	VAR robtarget Openhole_5522 := [[482.14, -9.61, 178.45], [0.078704, 0.702713, 0.693768, -0.136696], [0,0,0,0], [9E9, 9E9, 9E9, 9E9, 9E9, 9E9]];
	VAR robtarget Openhole_5523 := [[481.64, -9.62, 178.5], [0.077135, 0.702887, 0.694058, -0.135217], [0,0,0,0], [9E9, 9E9, 9E9, 9E9, 9E9, 9E9]];
	VAR robtarget Openhole_5524 := [[476.67, -9.77, 178.99], [0.061718, 0.704408, 0.696901, -0.119702], [0,0,0,0], [9E9, 9E9, 9E9, 9E9, 9E9, 9E9]];
	VAR robtarget Openhole_5525 := [[472.72, -10.2, 179.44], [0.050233, 0.70532, 0.699112, -0.106028], [0,0,0,0], [9E9, 9E9, 9E9, 9E9, 9E9, 9E9]];
	VAR robtarget Openhole_5526 := [[469.79, -10.75, 179.79], [0.042383, 0.705835, 0.700704, -0.094942], [0,0,0,0], [9E9, 9E9, 9E9, 9E9, 9E9, 9E9]];
	VAR robtarget Openhole_5527 := [[466.45, -11.71, 180.22], [0.034434, 0.706268, 0.702451, -0.081013], [0,0,0,0], [9E9, 9E9, 9E9, 9E9, 9E9, 9E9]];
	VAR robtarget Openhole_5528 := [[465.52, -12.04, 180.33], [0.0324, 0.706364, 0.702917, -0.076862], [0,0,0,0], [9E9, 9E9, 9E9, 9E9, 9E9, 9E9]];
	VAR robtarget Openhole_5529 := [[465.05, -12.22, 180.39], [0.031455, 0.706407, 0.703145, -0.074747], [0,0,0,0], [9E9, 9E9, 9E9, 9E9, 9E9, 9E9]];
	VAR robtarget Openhole_5530 := [[463.68, -12.81, 180.56], [0.028831, 0.706519, 0.703802, -0.068286], [0,0,0,0], [9E9, 9E9, 9E9, 9E9, 9E9, 9E9]];
	VAR robtarget Openhole_5531 := [[463.23, -13.02, 180.62], [0.028028, 0.706551, 0.704011, -0.066095], [0,0,0,0], [9E9, 9E9, 9E9, 9E9, 9E9, 9E9]];
	VAR robtarget Openhole_5532 := [[461.04, -14.18, 180.88], [0.024524, 0.706681, 0.704972, -0.05491], [0,0,0,0], [9E9, 9E9, 9E9, 9E9, 9E9, 9E9]];
	VAR robtarget Openhole_5533 := [[460.18, -14.69, 180.97], [0.023348, 0.706721, 0.705312, -0.050345], [0,0,0,0], [9E9, 9E9, 9E9, 9E9, 9E9, 9E9]];
	VAR robtarget Openhole_5534 := [[459.34, -15.23, 181.06], [0.022345, 0.706754, 0.705627, -0.045724], [0,0,0,0], [9E9, 9E9, 9E9, 9E9, 9E9, 9E9]];
	VAR robtarget Openhole_5535 := [[458.92, -15.49, 181.1], [0.021792, 0.706771, 0.705772, -0.04342], [0,0,0,0], [9E9, 9E9, 9E9, 9E9, 9E9, 9E9]];
	VAR robtarget Openhole_5536 := [[458.49, -15.74, 181.13], [0.021166, 0.70679, 0.70591, -0.041131], [0,0,0,0], [9E9, 9E9, 9E9, 9E9, 9E9, 9E9]];
	VAR robtarget Openhole_5537 := [[457.6, -16.2, 181.2], [0.019722, 0.706832, 0.706159, -0.036599], [0,0,0,0], [9E9, 9E9, 9E9, 9E9, 9E9, 9E9]];
	VAR robtarget Openhole_5538 := [[457.02, -16.45, 181.23], [0.018633, 0.706861, 0.706298, -0.033803], [0,0,0,0], [9E9, 9E9, 9E9, 9E9, 9E9, 9E9]];
	VAR robtarget Openhole_5539 := [[454.58, -16.45, 181.29], [0.010319, 0.707031, 0.706646, -0.025537], [0,0,0,0], [9E9, 9E9, 9E9, 9E9, 9E9, 9E9]];
	VAR robtarget Openhole_5540 := [[454.01, -15.03, 181.24], [0.003545, 0.707098, 0.706535, -0.028428], [0,0,0,0], [9E9, 9E9, 9E9, 9E9, 9E9, 9E9]];
	VAR robtarget Openhole_5541 := [[456.45, -15.03, 181.15], [0.011872, 0.707007, 0.706154, -0.036692], [0,0,0,0], [9E9, 9E9, 9E9, 9E9, 9E9, 9E9]];
	VAR robtarget Openhole_5542 := [[457.91, -14.13, 181.02], [0.013741, 0.706973, 0.705696, -0.044638], [0,0,0,0], [9E9, 9E9, 9E9, 9E9, 9E9, 9E9]];
	VAR robtarget Openhole_5543 := [[458.76, -13.61, 180.93], [0.014897, 0.70695, 0.705391, -0.049232], [0,0,0,0], [9E9, 9E9, 9E9, 9E9, 9E9, 9E9]];
	VAR robtarget Openhole_5544 := [[459.2, -13.37, 180.89], [0.015574, 0.706935, 0.705229, -0.051497], [0,0,0,0], [9E9, 9E9, 9E9, 9E9, 9E9, 9E9]];
	VAR robtarget Openhole_5545 := [[459.64, -13.14, 180.84], [0.016297, 0.706919, 0.705061, -0.053745], [0,0,0,0], [9E9, 9E9, 9E9, 9E9, 9E9, 9E9]];
	VAR robtarget Openhole_5546 := [[460.54, -12.71, 180.74], [0.017862, 0.706881, 0.704708, -0.05819], [0,0,0,0], [9E9, 9E9, 9E9, 9E9, 9E9, 9E9]];
	VAR robtarget Openhole_5547 := [[461.9, -12.1, 180.58], [0.020434, 0.706811, 0.704136, -0.064748], [0,0,0,0], [9E9, 9E9, 9E9, 9E9, 9E9, 9E9]];
	VAR robtarget Openhole_5548 := [[463.74, -11.36, 180.36], [0.024178, 0.706693, 0.703297, -0.073302], [0,0,0,0], [9E9, 9E9, 9E9, 9E9, 9E9, 9E9]];
	VAR robtarget Openhole_5549 := [[466.57, -10.43, 180], [0.030537, 0.706447, 0.701901, -0.085647], [0,0,0,0], [9E9, 9E9, 9E9, 9E9, 9E9, 9E9]];
	VAR robtarget Openhole_5550 := [[468.97, -9.8, 179.68], [0.036475, 0.706165, 0.700635, -0.095449], [0,0,0,0], [9E9, 9E9, 9E9, 9E9, 9E9, 9E9]];
	VAR robtarget Openhole_5551 := [[472.87, -9.09, 179.17], [0.047062, 0.705539, 0.698476, -0.110139], [0,0,0,0], [9E9, 9E9, 9E9, 9E9, 9E9, 9E9]];
	VAR robtarget Openhole_5552 := [[477.32, -8.67, 178.63], [0.060222, 0.704538, 0.695928, -0.125238], [0,0,0,0], [9E9, 9E9, 9E9, 9E9, 9E9, 9E9]];
	VAR robtarget Openhole_5553 := [[481.79, -8.56, 178.15], [0.074227, 0.7032, 0.693312, -0.13899], [0,0,0,0], [9E9, 9E9, 9E9, 9E9, 9E9, 9E9]];
	VAR robtarget Openhole_5554 := [[482.29, -8.56, 178.1], [0.075808, 0.703031, 0.693017, -0.140454], [0,0,0,0], [9E9, 9E9, 9E9, 9E9, 9E9, 9E9]];
	VAR robtarget Openhole_5555 := [[490.75, -8.89, 177.38], [0.102945, 0.699573, 0.687924, -0.163586], [0,0,0,0], [9E9, 9E9, 9E9, 9E9, 9E9, 9E9]];
	VAR robtarget Openhole_5556 := [[499.22, -9.25, 176.73], [0.128731, 0.69529, 0.682463, -0.185054], [0,0,0,0], [9E9, 9E9, 9E9, 9E9, 9E9, 9E9]];
	VAR robtarget Openhole_5557 := [[500.21, -9.26, 176.64], [0.131553, 0.694762, 0.681773, -0.187578], [0,0,0,0], [9E9, 9E9, 9E9, 9E9, 9E9, 9E9]];
	VAR robtarget Openhole_5558 := [[500.71, -9.26, 176.59], [0.132933, 0.694499, 0.681421, -0.188853], [0,0,0,0], [9E9, 9E9, 9E9, 9E9, 9E9, 9E9]];
	VAR robtarget Openhole_5559 := [[503.19, -9.2, 176.33], [0.139644, 0.693181, 0.679622, -0.195227], [0,0,0,0], [9E9, 9E9, 9E9, 9E9, 9E9, 9E9]];
	VAR robtarget Openhole_5560 := [[503.69, -9.17, 176.27], [0.1409, 0.692927, 0.679243, -0.196542], [0,0,0,0], [9E9, 9E9, 9E9, 9E9, 9E9, 9E9]];
	VAR robtarget Openhole_5561 := [[504.33, -9.15, 176.19], [0.142564, 0.692586, 0.678764, -0.198192], [0,0,0,0], [9E9, 9E9, 9E9, 9E9, 9E9, 9E9]];
	VAR robtarget Openhole_5562 := [[509.33, -9.15, 175.72], [0.183051, 0.683002, 0.683002, -0.183051], [0,0,0,0], [9E9, 9E9, 9E9, 9E9, 9E9, 9E9]];
	VAR robtarget Openhole_5563 := [[536.33, -9.15, 175.63], [0.183051, 0.683002, 0.683002, -0.183051], [0,0,0,0], [9E9, 9E9, 9E9, 9E9, 9E9, 9E9]];
	VAR robtarget Openhole_5564 := [[536.33, -8.27, 175.13], [0.183051, 0.683002, 0.683002, -0.183051], [0,0,0,0], [9E9, 9E9, 9E9, 9E9, 9E9, 9E9]];
	VAR robtarget Openhole_5565 := [[524.33, -8.27, 175.17], [0.183051, 0.683002, 0.683002, -0.183051], [0,0,0,0], [9E9, 9E9, 9E9, 9E9, 9E9, 9E9]];
	VAR robtarget Openhole_5566 := [[509.33, -8.28, 175.21], [0.183051, 0.683002, 0.683002, -0.183051], [0,0,0,0], [9E9, 9E9, 9E9, 9E9, 9E9, 9E9]];
	VAR robtarget Openhole_5567 := [[504.35, -8.28, 175.73], [0.140085, 0.693092, 0.678014, -0.20074], [0,0,0,0], [9E9, 9E9, 9E9, 9E9, 9E9, 9E9]];
	VAR robtarget Openhole_5568 := [[503.83, -8.3, 175.8], [0.138746, 0.693361, 0.678412, -0.199393], [0,0,0,0], [9E9, 9E9, 9E9, 9E9, 9E9, 9E9]];
	VAR robtarget Openhole_5569 := [[501.35, -8.33, 176.06], [0.131956, 0.694685, 0.68021, -0.193171], [0,0,0,0], [9E9, 9E9, 9E9, 9E9, 9E9, 9E9]];
	VAR robtarget Openhole_5570 := [[500.85, -8.32, 176.11], [0.13055, 0.694951, 0.680559, -0.191937], [0,0,0,0], [9E9, 9E9, 9E9, 9E9, 9E9, 9E9]];
	VAR robtarget Openhole_5571 := [[493.88, -7.98, 176.68], [0.10947, 0.698582, 0.685143, -0.174867], [0,0,0,0], [9E9, 9E9, 9E9, 9E9, 9E9, 9E9]];
	VAR robtarget Openhole_5572 := [[483.94, -7.4, 177.55], [0.077321, 0.702867, 0.691248, -0.148916], [0,0,0,0], [9E9, 9E9, 9E9, 9E9, 9E9, 9E9]];
	VAR robtarget Openhole_5573 := [[480.96, -7.35, 177.87], [0.0677, 0.703858, 0.69304, -0.140343], [0,0,0,0], [9E9, 9E9, 9E9, 9E9, 9E9, 9E9]];
	VAR robtarget Openhole_5574 := [[480.46, -7.35, 177.92], [0.066114, 0.704009, 0.693337, -0.138866], [0,0,0,0], [9E9, 9E9, 9E9, 9E9, 9E9, 9E9]];
	VAR robtarget Openhole_5575 := [[476, -7.51, 178.47], [0.052157, 0.705181, 0.695985, -0.12492], [0,0,0,0], [9E9, 9E9, 9E9, 9E9, 9E9, 9E9]];
	VAR robtarget Openhole_5576 := [[471.56, -7.98, 179.06], [0.039093, 0.706025, 0.698557, -0.109628], [0,0,0,0], [9E9, 9E9, 9E9, 9E9, 9E9, 9E9]];
	VAR robtarget Openhole_5577 := [[467.18, -8.8, 179.67], [0.027176, 0.706584, 0.700967, -0.092983], [0,0,0,0], [9E9, 9E9, 9E9, 9E9, 9E9, 9E9]];
	VAR robtarget Openhole_5578 := [[464.77, -9.39, 179.99], [0.021046, 0.706794, 0.702192, -0.083224], [0,0,0,0], [9E9, 9E9, 9E9, 9E9, 9E9, 9E9]];
	VAR robtarget Openhole_5579 := [[459.06, -11.07, 180.68], [0.007315, 0.707069, 0.704662, -0.058745], [0,0,0,0], [9E9, 9E9, 9E9, 9E9, 9E9, 9E9]];
	VAR robtarget Openhole_5580 := [[458.11, -11.38, 180.78], [0.005116, 0.707088, 0.704999, -0.05456], [0,0,0,0], [9E9, 9E9, 9E9, 9E9, 9E9, 9E9]];
	VAR robtarget Openhole_5581 := [[457.17, -11.7, 180.87], [0.00302, 0.7071, 0.705315, -0.05031], [0,0,0,0], [9E9, 9E9, 9E9, 9E9, 9E9, 9E9]];
	VAR robtarget Openhole_5582 := [[456.7, -11.89, 180.92], [0.002058, 0.707104, 0.705466, -0.048142], [0,0,0,0], [9E9, 9E9, 9E9, 9E9, 9E9, 9E9]];
	VAR robtarget Openhole_5583 := [[456.25, -12.09, 180.96], [0.001205, 0.707106, 0.705614, -0.045926], [0,0,0,0], [9E9, 9E9, 9E9, 9E9, 9E9, 9E9]];
	VAR robtarget Openhole_5584 := [[455.8, -12.3, 181], [0.000391, 0.707107, 0.705756, -0.043694], [0,0,0,0], [9E9, 9E9, 9E9, 9E9, 9E9, 9E9]];
	VAR robtarget Openhole_5585 := [[455.36, -12.53, 181.05], [-0.000349, 0.707107, 0.705892, -0.041433], [0,0,0,0], [9E9, 9E9, 9E9, 9E9, 9E9, 9E9]];
	VAR robtarget Openhole_5586 := [[454.83, -12.87, 181.1], [-0.001006, 0.707106, 0.706058, -0.038495], [0,0,0,0], [9E9, 9E9, 9E9, 9E9, 9E9, 9E9]];
	VAR robtarget Openhole_5587 := [[445.25, -11.83, 181.71], [-0.03715, 0.70613, 0.707042, -0.009558], [0,0,0,0], [9E9, 9E9, 9E9, 9E9, 9E9, 9E9]];
	VAR robtarget Openhole_5588 := [[444.72, -11.69, 181.75], [-0.039438, 0.706006, 0.707059, -0.008218], [0,0,0,0], [9E9, 9E9, 9E9, 9E9, 9E9, 9E9]];
	VAR robtarget Openhole_5589 := [[444.22, -11.62, 181.79], [-0.041326, 0.705898, 0.707075, -0.006749], [0,0,0,0], [9E9, 9E9, 9E9, 9E9, 9E9, 9E9]];
	VAR robtarget Openhole_5590 := [[443.23, -11.52, 181.86], [-0.045015, 0.705673, 0.707097, -0.003709], [0,0,0,0], [9E9, 9E9, 9E9, 9E9, 9E9, 9E9]];
	VAR robtarget Openhole_5591 := [[442.24, -11.45, 181.94], [-0.048615, 0.705434, 0.707107, -0.000574], [0,0,0,0], [9E9, 9E9, 9E9, 9E9, 9E9, 9E9]];
	VAR robtarget Openhole_5592 := [[441.74, -11.43, 181.98], [-0.050381, 0.70531, 0.707106, 0.001028], [0,0,0,0], [9E9, 9E9, 9E9, 9E9, 9E9, 9E9]];
	VAR robtarget Openhole_5593 := [[431.77, -11.25, 182.74], [-0.08402, 0.702097, 0.706286, 0.03406], [0,0,0,0], [9E9, 9E9, 9E9, 9E9, 9E9, 9E9]];
	VAR robtarget Openhole_5594 := [[431.27, -11.25, 182.77], [-0.085634, 0.701902, 0.706204, 0.035729], [0,0,0,0], [9E9, 9E9, 9E9, 9E9, 9E9, 9E9]];
	VAR robtarget Openhole_5595 := [[407.33, -11.81, 184.34], [-0.156518, 0.689567, 0.697978, 0.113254], [0,0,0,0], [9E9, 9E9, 9E9, 9E9, 9E9, 9E9]];
	VAR robtarget Openhole_5596 := [[396.35, -12.23, 184.89], [-0.184529, 0.682605, 0.69195, 0.145619], [0,0,0,0], [9E9, 9E9, 9E9, 9E9, 9E9, 9E9]];
	VAR robtarget Openhole_5597 := [[394.34, -12.34, 184.96], [-0.189276, 0.681304, 0.690716, 0.151363], [0,0,0,0], [9E9, 9E9, 9E9, 9E9, 9E9, 9E9]];
	VAR robtarget Openhole_5598 := [[389.36, -12.34, 185.28], [-0.201409, 0.677816, 0.687741, 0.164354], [0,0,0,0], [9E9, 9E9, 9E9, 9E9, 9E9, 9E9]];
	VAR robtarget Openhole_5599 := [[362.36, -12.34, 185.37], [-0.183051, 0.683002, 0.683002, 0.183051], [0,0,0,0], [9E9, 9E9, 9E9, 9E9, 9E9, 9E9]];
	VAR robtarget Openhole_5600 := [[362.36, -13.23, 184.86], [-0.183051, 0.683002, 0.683002, 0.183051], [0,0,0,0], [9E9, 9E9, 9E9, 9E9, 9E9, 9E9]];
	VAR robtarget Openhole_5601 := [[374.36, -13.23, 184.82], [-0.183051, 0.683002, 0.683002, 0.183051], [0,0,0,0], [9E9, 9E9, 9E9, 9E9, 9E9, 9E9]];
	VAR robtarget Openhole_5602 := [[389.36, -13.23, 184.77], [-0.198916, 0.678552, 0.687133, 0.166878], [0,0,0,0], [9E9, 9E9, 9E9, 9E9, 9E9, 9E9]];
	VAR robtarget Openhole_5603 := [[394.33, -13.23, 184.49], [-0.186724, 0.682007, 0.690143, 0.153955], [0,0,0,0], [9E9, 9E9, 9E9, 9E9, 9E9, 9E9]];
	VAR robtarget Openhole_5604 := [[404.34, -12.8, 184.12], [-0.161764, 0.688355, 0.695969, 0.125011], [0,0,0,0], [9E9, 9E9, 9E9, 9E9, 9E9, 9E9]];
	VAR robtarget Openhole_5605 := [[421.81, -12.49, 183.16], [-0.111659, 0.698235, 0.703558, 0.070753], [0,0,0,0], [9E9, 9E9, 9E9, 9E9, 9E9, 9E9]];
	VAR robtarget Openhole_5606 := [[427.8, -12.45, 182.78], [-0.092876, 0.700981, 0.70525, 0.051205], [0,0,0,0], [9E9, 9E9, 9E9, 9E9, 9E9, 9E9]];
	VAR robtarget Openhole_5607 := [[428.3, -12.46, 182.75], [-0.09127, 0.701192, 0.705367, 0.049569], [0,0,0,0], [9E9, 9E9, 9E9, 9E9, 9E9, 9E9]];
	VAR robtarget Openhole_5608 := [[434.78, -12.62, 182.32], [-0.069589, 0.703674, 0.70653, 0.028563], [0,0,0,0], [9E9, 9E9, 9E9, 9E9, 9E9, 9E9]];
	VAR robtarget Openhole_5609 := [[440.25, -13.05, 181.95], [-0.049924, 0.705342, 0.707013, 0.011547], [0,0,0,0], [9E9, 9E9, 9E9, 9E9, 9E9, 9E9]];
	VAR robtarget Openhole_5610 := [[442.74, -13.1, 181.8], [-0.041319, 0.705899, 0.707099, 0.003283], [0,0,0,0], [9E9, 9E9, 9E9, 9E9, 9E9, 9E9]];
	VAR robtarget Openhole_5611 := [[443.44, -13.31, 181.75], [-0.038283, 0.70607, 0.707105, 0.001638], [0,0,0,0], [9E9, 9E9, 9E9, 9E9, 9E9, 9E9]];
	VAR robtarget Openhole_5612 := [[445.21, -13.31, 181.65], [-0.03227, 0.70637, 0.707093, -0.004388], [0,0,0,0], [9E9, 9E9, 9E9, 9E9, 9E9, 9E9]];
	VAR robtarget Openhole_5613 := [[444.28, -14.54, 181.64], [-0.031215, 0.706417, 0.707101, 0.002931], [0,0,0,0], [9E9, 9E9, 9E9, 9E9, 9E9, 9E9]];
	VAR robtarget Openhole_5614 := [[442.51, -14.54, 181.72], [-0.037224, 0.706126, 0.70705, 0.008951], [0,0,0,0], [9E9, 9E9, 9E9, 9E9, 9E9, 9E9]];
	VAR robtarget Openhole_5615 := [[441.98, -14.53, 181.74], [-0.039072, 0.706026, 0.707026, 0.010719], [0,0,0,0], [9E9, 9E9, 9E9, 9E9, 9E9, 9E9]];
	VAR robtarget Openhole_5616 := [[440.98, -14.49, 181.79], [-0.042583, 0.705823, 0.706969, 0.013957], [0,0,0,0], [9E9, 9E9, 9E9, 9E9, 9E9, 9E9]];
	VAR robtarget Openhole_5617 := [[439.98, -14.49, 181.83], [-0.045964, 0.705611, 0.706895, 0.017319], [0,0,0,0], [9E9, 9E9, 9E9, 9E9, 9E9, 9E9]];
	VAR robtarget Openhole_5618 := [[439.48, -14.47, 181.85], [-0.04768, 0.705497, 0.706852, 0.01897], [0,0,0,0], [9E9, 9E9, 9E9, 9E9, 9E9, 9E9]];
	VAR robtarget Openhole_5619 := [[438.98, -14.45, 181.88], [-0.049444, 0.705376, 0.706808, 0.020564], [0,0,0,0], [9E9, 9E9, 9E9, 9E9, 9E9, 9E9]];
	VAR robtarget Openhole_5620 := [[438.48, -14.4, 181.9], [-0.051258, 0.705247, 0.706761, 0.022097], [0,0,0,0], [9E9, 9E9, 9E9, 9E9, 9E9, 9E9]];
	VAR robtarget Openhole_5621 := [[433.03, -13.83, 182.24], [-0.071327, 0.7035, 0.70606, 0.038469], [0,0,0,0], [9E9, 9E9, 9E9, 9E9, 9E9, 9E9]];
	VAR robtarget Openhole_5622 := [[426.54, -13.59, 182.61], [-0.093145, 0.700945, 0.704635, 0.05907], [0,0,0,0], [9E9, 9E9, 9E9, 9E9, 9E9, 9E9]];
	VAR robtarget Openhole_5623 := [[419.55, -13.55, 182.99], [-0.115196, 0.69766, 0.702409, 0.08137], [0,0,0,0], [9E9, 9E9, 9E9, 9E9, 9E9, 9E9]];
	VAR robtarget Openhole_5624 := [[419.05, -13.55, 183.02], [-0.116726, 0.697406, 0.702225, 0.082945], [0,0,0,0], [9E9, 9E9, 9E9, 9E9, 9E9, 9E9]];
	VAR robtarget Openhole_5625 := [[404.07, -13.73, 183.73], [-0.159674, 0.688843, 0.695311, 0.128617], [0,0,0,0], [9E9, 9E9, 9E9, 9E9, 9E9, 9E9]];
	VAR robtarget Openhole_5626 := [[394.35, -14.11, 184.02], [-0.18411, 0.682718, 0.689575, 0.156483], [0,0,0,0], [9E9, 9E9, 9E9, 9E9, 9E9, 9E9]];
	VAR robtarget Openhole_5627 := [[389.36, -14.11, 184.26], [-0.19642, 0.679279, 0.686516, 0.1694], [0,0,0,0], [9E9, 9E9, 9E9, 9E9, 9E9, 9E9]];
	VAR robtarget Openhole_5628 := [[362.36, -14.11, 184.35], [-0.183051, 0.683002, 0.683002, 0.183051], [0,0,0,0], [9E9, 9E9, 9E9, 9E9, 9E9, 9E9]];
	VAR robtarget Openhole_5629 := [[362.35, -15.07, 183.79], [-0.183051, 0.683002, 0.683002, 0.183051], [0,0,0,0], [9E9, 9E9, 9E9, 9E9, 9E9, 9E9]];
	VAR robtarget Openhole_5630 := [[389.35, -15.07, 183.7], [-0.193687, 0.680063, 0.68583, 0.172155], [0,0,0,0], [9E9, 9E9, 9E9, 9E9, 9E9, 9E9]];
	VAR robtarget Openhole_5631 := [[394.35, -15.07, 183.51], [-0.181307, 0.683467, 0.688928, 0.159306], [0,0,0,0], [9E9, 9E9, 9E9, 9E9, 9E9, 9E9]];
	VAR robtarget Openhole_5632 := [[404.04, -14.7, 183.31], [-0.15678, 0.689507, 0.694738, 0.131678], [0,0,0,0], [9E9, 9E9, 9E9, 9E9, 9E9, 9E9]];
	VAR robtarget Openhole_5633 := [[413.54, -14.6, 182.95], [-0.12998, 0.695058, 0.699507, 0.10339], [0,0,0,0], [9E9, 9E9, 9E9, 9E9, 9E9, 9E9]];
	VAR robtarget Openhole_5634 := [[414.04, -14.6, 182.93], [-0.128498, 0.695333, 0.69973, 0.101869], [0,0,0,0], [9E9, 9E9, 9E9, 9E9, 9E9, 9E9]];
	VAR robtarget Openhole_5635 := [[427.52, -14.77, 182.32], [-0.086129, 0.701842, 0.704577, 0.059757], [0,0,0,0], [9E9, 9E9, 9E9, 9E9, 9E9, 9E9]];
	VAR robtarget Openhole_5636 := [[434, -15.12, 182], [-0.063775, 0.704225, 0.706, 0.039544], [0,0,0,0], [9E9, 9E9, 9E9, 9E9, 9E9, 9E9]];
	VAR robtarget Openhole_5637 := [[437.48, -15.49, 181.83], [-0.050954, 0.705269, 0.706505, 0.029156], [0,0,0,0], [9E9, 9E9, 9E9, 9E9, 9E9, 9E9]];
	VAR robtarget Openhole_5638 := [[438.47, -15.58, 181.78], [-0.047326, 0.705521, 0.706625, 0.026099], [0,0,0,0], [9E9, 9E9, 9E9, 9E9, 9E9, 9E9]];
	VAR robtarget Openhole_5639 := [[438.97, -15.61, 181.76], [-0.045564, 0.705637, 0.706682, 0.024503], [0,0,0,0], [9E9, 9E9, 9E9, 9E9, 9E9, 9E9]];
	VAR robtarget Openhole_5640 := [[439.47, -15.62, 181.75], [-0.043835, 0.705747, 0.706737, 0.022869], [0,0,0,0], [9E9, 9E9, 9E9, 9E9, 9E9, 9E9]];
	VAR robtarget Openhole_5641 := [[439.97, -15.62, 181.73], [-0.04214, 0.70585, 0.706789, 0.021196], [0,0,0,0], [9E9, 9E9, 9E9, 9E9, 9E9, 9E9]];
	VAR robtarget Openhole_5642 := [[440.97, -15.59, 181.7], [-0.038871, 0.706038, 0.706885, 0.01772], [0,0,0,0], [9E9, 9E9, 9E9, 9E9, 9E9, 9E9]];
	VAR robtarget Openhole_5643 := [[441.46, -15.51, 181.69], [-0.0375, 0.706112, 0.706931, 0.015763], [0,0,0,0], [9E9, 9E9, 9E9, 9E9, 9E9, 9E9]];
	VAR robtarget Openhole_5644 := [[442.03, -15.46, 181.67], [-0.035743, 0.706203, 0.706975, 0.013654], [0,0,0,0], [9E9, 9E9, 9E9, 9E9, 9E9, 9E9]];
	VAR robtarget Openhole_5645 := [[443.93, -15.46, 181.61], [-0.029319, 0.706499, 0.70707, 0.007225], [0,0,0,0], [9E9, 9E9, 9E9, 9E9, 9E9, 9E9]];
	VAR robtarget Openhole_5646 := [[443.56, -16.48, 181.56], [-0.027098, 0.706587, 0.707005, 0.011974], [0,0,0,0], [9E9, 9E9, 9E9, 9E9, 9E9, 9E9]];
	VAR robtarget Openhole_5647 := [[441.66, -16.48, 181.61], [-0.033523, 0.706312, 0.706867, 0.018395], [0,0,0,0], [9E9, 9E9, 9E9, 9E9, 9E9, 9E9]];
	VAR robtarget Openhole_5648 := [[441.11, -16.58, 181.62], [-0.035051, 0.706238, 0.706808, 0.020566], [0,0,0,0], [9E9, 9E9, 9E9, 9E9, 9E9, 9E9]];
	VAR robtarget Openhole_5649 := [[440.63, -16.69, 181.62], [-0.036318, 0.706173, 0.706746, 0.02259], [0,0,0,0], [9E9, 9E9, 9E9, 9E9, 9E9, 9E9]];
	VAR robtarget Openhole_5650 := [[440.13, -16.73, 181.63], [-0.037867, 0.706092, 0.706686, 0.024405], [0,0,0,0], [9E9, 9E9, 9E9, 9E9, 9E9, 9E9]];
	VAR robtarget Openhole_5651 := [[438.63, -16.79, 181.65], [-0.042721, 0.705815, 0.706485, 0.029646], [0,0,0,0], [9E9, 9E9, 9E9, 9E9, 9E9, 9E9]];
	VAR robtarget Openhole_5652 := [[437.63, -16.79, 181.67], [-0.046068, 0.705605, 0.706336, 0.033016], [0,0,0,0], [9E9, 9E9, 9E9, 9E9, 9E9, 9E9]];
	VAR robtarget Openhole_5653 := [[437.13, -16.79, 181.68], [-0.047751, 0.705493, 0.706256, 0.034685], [0,0,0,0], [9E9, 9E9, 9E9, 9E9, 9E9, 9E9]];
	VAR robtarget Openhole_5654 := [[414.15, -16.27, 182.36], [-0.122868, 0.69635, 0.698989, 0.106841], [0,0,0,0], [9E9, 9E9, 9E9, 9E9, 9E9, 9E9]];
	VAR robtarget Openhole_5655 := [[410.15, -16.25, 182.47], [-0.134734, 0.694152, 0.697065, 0.118744], [0,0,0,0], [9E9, 9E9, 9E9, 9E9, 9E9, 9E9]];
	VAR robtarget Openhole_5656 := [[409.65, -16.25, 182.48], [-0.136184, 0.693869, 0.696812, 0.120219], [0,0,0,0], [9E9, 9E9, 9E9, 9E9, 9E9, 9E9]];
	VAR robtarget Openhole_5657 := [[399.65, -16.42, 182.67], [-0.163515, 0.687941, 0.691204, 0.149119], [0,0,0,0], [9E9, 9E9, 9E9, 9E9, 9E9, 9E9]];
	VAR robtarget Openhole_5658 := [[395.16, -16.63, 182.67], [-0.174709, 0.685184, 0.688357, 0.161754], [0,0,0,0], [9E9, 9E9, 9E9, 9E9, 9E9, 9E9]];
	VAR robtarget Openhole_5659 := [[394.35, -16.66, 182.67], [-0.176688, 0.684676, 0.687838, 0.163946], [0,0,0,0], [9E9, 9E9, 9E9, 9E9, 9E9, 9E9]];
	VAR robtarget Openhole_5660 := [[389.35, -16.66, 182.79], [-0.189184, 0.681329, 0.684678, 0.176681], [0,0,0,0], [9E9, 9E9, 9E9, 9E9, 9E9, 9E9]];
	VAR robtarget Openhole_5661 := [[362.35, -16.66, 182.87], [-0.183051, 0.683002, 0.683002, 0.183051], [0,0,0,0], [9E9, 9E9, 9E9, 9E9, 9E9, 9E9]];
	VAR robtarget Openhole_5662 := [[362.34, -19.81, 181.05], [-0.183051, 0.683002, 0.683002, 0.183051], [0,0,0,0], [9E9, 9E9, 9E9, 9E9, 9E9, 9E9]];
	VAR robtarget Openhole_5663 := [[389.34, -19.81, 180.97], [-0.180222, 0.683754, 0.682302, 0.185644], [0,0,0,0], [9E9, 9E9, 9E9, 9E9, 9E9, 9E9]];
	VAR robtarget Openhole_5664 := [[394.34, -19.81, 181.01], [-0.167496, 0.686983, 0.685583, 0.173136], [0,0,0,0], [9E9, 9E9, 9E9, 9E9, 9E9, 9E9]];
	VAR robtarget Openhole_5665 := [[402.02, -19.48, 181.21], [-0.147838, 0.69148, 0.69061, 0.151848], [0,0,0,0], [9E9, 9E9, 9E9, 9E9, 9E9, 9E9]];
	VAR robtarget Openhole_5666 := [[407.52, -19.42, 181.26], [-0.13245, 0.694591, 0.693853, 0.136265], [0,0,0,0], [9E9, 9E9, 9E9, 9E9, 9E9, 9E9]];
	VAR robtarget Openhole_5667 := [[408.02, -19.42, 181.26], [-0.131, 0.694866, 0.694132, 0.134834], [0,0,0,0], [9E9, 9E9, 9E9, 9E9, 9E9, 9E9]];
	VAR robtarget Openhole_5668 := [[422.52, -19.62, 181.27], [-0.086168, 0.701837, 0.701129, 0.091747], [0,0,0,0], [9E9, 9E9, 9E9, 9E9, 9E9, 9E9]];
	VAR robtarget Openhole_5669 := [[423.02, -19.61, 181.27], [-0.084577, 0.70203, 0.701334, 0.090169], [0,0,0,0], [9E9, 9E9, 9E9, 9E9, 9E9, 9E9]];
	VAR robtarget Openhole_5670 := [[428.01, -19.47, 181.33], [-0.068925, 0.70374, 0.703253, 0.073721], [0,0,0,0], [9E9, 9E9, 9E9, 9E9, 9E9, 9E9]];
	VAR robtarget Openhole_5671 := [[429.01, -19.4, 181.35], [-0.065889, 0.70403, 0.703607, 0.070262], [0,0,0,0], [9E9, 9E9, 9E9, 9E9, 9E9, 9E9]];
	VAR robtarget Openhole_5672 := [[429.51, -19.35, 181.36], [-0.064414, 0.704167, 0.703782, 0.068487], [0,0,0,0], [9E9, 9E9, 9E9, 9E9, 9E9, 9E9]];
	VAR robtarget Openhole_5673 := [[430.5, -19.24, 181.38], [-0.061526, 0.704425, 0.704125, 0.064869], [0,0,0,0], [9E9, 9E9, 9E9, 9E9, 9E9, 9E9]];
	VAR robtarget Openhole_5674 := [[433.97, -18.76, 181.46], [-0.051674, 0.705216, 0.705204, 0.051842], [0,0,0,0], [9E9, 9E9, 9E9, 9E9, 9E9, 9E9]];
	VAR robtarget Openhole_5675 := [[434.46, -18.67, 181.47], [-0.050313, 0.705315, 0.705342, 0.049927], [0,0,0,0], [9E9, 9E9, 9E9, 9E9, 9E9, 9E9]];
	VAR robtarget Openhole_5676 := [[434.95, -18.6, 181.48], [-0.048909, 0.705413, 0.705473, 0.048039], [0,0,0,0], [9E9, 9E9, 9E9, 9E9, 9E9, 9E9]];
	VAR robtarget Openhole_5677 := [[435.94, -18.42, 181.5], [-0.046239, 0.705593, 0.705727, 0.044153], [0,0,0,0], [9E9, 9E9, 9E9, 9E9, 9E9, 9E9]];
	VAR robtarget Openhole_5678 := [[436.43, -18.34, 181.51], [-0.044854, 0.705683, 0.705844, 0.042239], [0,0,0,0], [9E9, 9E9, 9E9, 9E9, 9E9, 9E9]];
	VAR robtarget Openhole_5679 := [[436.92, -18.24, 181.52], [-0.043539, 0.705765, 0.705959, 0.040273], [0,0,0,0], [9E9, 9E9, 9E9, 9E9, 9E9, 9E9]];
	VAR robtarget Openhole_5680 := [[440.87, -17.63, 181.54], [-0.032306, 0.706368, 0.706668, 0.024919], [0,0,0,0], [9E9, 9E9, 9E9, 9E9, 9E9, 9E9]];
	VAR robtarget Openhole_5681 := [[441.37, -17.54, 181.54], [-0.030927, 0.70643, 0.706734, 0.022968], [0,0,0,0], [9E9, 9E9, 9E9, 9E9, 9E9, 9E9]];
	VAR robtarget Openhole_5682 := [[441.43, -17.55, 181.53], [-0.03068, 0.706441, 0.70674, 0.022783], [0,0,0,0], [9E9, 9E9, 9E9, 9E9, 9E9, 9E9]];
	VAR robtarget Openhole_5683 := [[443.2, -17.55, 181.51], [-0.024666, 0.706676, 0.706908, 0.016783], [0,0,0,0], [9E9, 9E9, 9E9, 9E9, 9E9, 9E9]];
	VAR robtarget Openhole_5684 := [[443.12, -18.53, 181.45], [-0.021596, 0.706777, 0.706813, 0.020397], [0,0,0,0], [9E9, 9E9, 9E9, 9E9, 9E9, 9E9]];
	VAR robtarget Openhole_5685 := [[441.35, -18.53, 181.46], [-0.027613, 0.706567, 0.706614, 0.026391], [0,0,0,0], [9E9, 9E9, 9E9, 9E9, 9E9, 9E9]];
	VAR robtarget Openhole_5686 := [[441.27, -18.53, 181.46], [-0.027878, 0.706557, 0.706605, 0.026645], [0,0,0,0], [9E9, 9E9, 9E9, 9E9, 9E9, 9E9]];
	VAR robtarget Openhole_5687 := [[440.77, -18.58, 181.46], [-0.029397, 0.706495, 0.706533, 0.028488], [0,0,0,0], [9E9, 9E9, 9E9, 9E9, 9E9, 9E9]];
	VAR robtarget Openhole_5688 := [[440.28, -18.68, 181.45], [-0.030733, 0.706439, 0.70645, 0.030465], [0,0,0,0], [9E9, 9E9, 9E9, 9E9, 9E9, 9E9]];
	VAR robtarget Openhole_5689 := [[439.31, -18.93, 181.43], [-0.033164, 0.706329, 0.706262, 0.03456], [0,0,0,0], [9E9, 9E9, 9E9, 9E9, 9E9, 9E9]];
	VAR robtarget Openhole_5690 := [[438.84, -19.07, 181.42], [-0.034287, 0.706275, 0.706156, 0.036656], [0,0,0,0], [9E9, 9E9, 9E9, 9E9, 9E9, 9E9]];
	VAR robtarget Openhole_5691 := [[438.36, -19.23, 181.4], [-0.035334, 0.706223, 0.706042, 0.038787], [0,0,0,0], [9E9, 9E9, 9E9, 9E9, 9E9, 9E9]];
	VAR robtarget Openhole_5692 := [[437.9, -19.41, 181.38], [-0.036284, 0.706175, 0.70592, 0.040959], [0,0,0,0], [9E9, 9E9, 9E9, 9E9, 9E9, 9E9]];
	VAR robtarget Openhole_5693 := [[436.99, -19.83, 181.33], [-0.037928, 0.706089, 0.705648, 0.045395], [0,0,0,0], [9E9, 9E9, 9E9, 9E9, 9E9, 9E9]];
	VAR robtarget Openhole_5694 := [[436.54, -20.05, 181.3], [-0.038715, 0.706046, 0.705501, 0.04762], [0,0,0,0], [9E9, 9E9, 9E9, 9E9, 9E9, 9E9]];
	VAR robtarget Openhole_5695 := [[436.1, -20.28, 181.26], [-0.039411, 0.706008, 0.705346, 0.049872], [0,0,0,0], [9E9, 9E9, 9E9, 9E9, 9E9, 9E9]];
	VAR robtarget Openhole_5696 := [[435.23, -20.76, 181.19], [-0.040708, 0.705934, 0.705012, 0.054389], [0,0,0,0], [9E9, 9E9, 9E9, 9E9, 9E9, 9E9]];
	VAR robtarget Openhole_5697 := [[434.78, -20.99, 181.15], [-0.041427, 0.705892, 0.704836, 0.056622], [0,0,0,0], [9E9, 9E9, 9E9, 9E9, 9E9, 9E9]];
	VAR robtarget Openhole_5698 := [[433.88, -21.41, 181.07], [-0.043028, 0.705796, 0.704469, 0.061017], [0,0,0,0], [9E9, 9E9, 9E9, 9E9, 9E9, 9E9]];
	VAR robtarget Openhole_5699 := [[432.49, -21.97, 180.94], [-0.045798, 0.705622, 0.703884, 0.067432], [0,0,0,0], [9E9, 9E9, 9E9, 9E9, 9E9, 9E9]];
	VAR robtarget Openhole_5700 := [[432.02, -22.13, 180.9], [-0.046808, 0.705556, 0.703681, 0.069523], [0,0,0,0], [9E9, 9E9, 9E9, 9E9, 9E9, 9E9]];
	VAR robtarget Openhole_5701 := [[430.6, -22.59, 180.78], [-0.049999, 0.705337, 0.703045, 0.075684], [0,0,0,0], [9E9, 9E9, 9E9, 9E9, 9E9, 9E9]];
	VAR robtarget Openhole_5702 := [[430.12, -22.73, 180.74], [-0.051125, 0.705256, 0.702825, 0.077695], [0,0,0,0], [9E9, 9E9, 9E9, 9E9, 9E9, 9E9]];
	VAR robtarget Openhole_5703 := [[428.19, -23.21, 180.57], [-0.055917, 0.704892, 0.701917, 0.085515], [0,0,0,0], [9E9, 9E9, 9E9, 9E9, 9E9, 9E9]];
	VAR robtarget Openhole_5704 := [[427.7, -23.31, 180.53], [-0.057184, 0.704791, 0.701683, 0.087414], [0,0,0,0], [9E9, 9E9, 9E9, 9E9, 9E9, 9E9]];
	VAR robtarget Openhole_5705 := [[426.72, -23.49, 180.45], [-0.059805, 0.704573, 0.701209, 0.091135], [0,0,0,0], [9E9, 9E9, 9E9, 9E9, 9E9, 9E9]];
	VAR robtarget Openhole_5706 := [[422.76, -23.95, 180.16], [-0.071176, 0.703515, 0.699252, 0.105104], [0,0,0,0], [9E9, 9E9, 9E9, 9E9, 9E9, 9E9]];
	VAR robtarget Openhole_5707 := [[417.27, -24.13, 179.85], [-0.088051, 0.701603, 0.696419, 0.122476], [0,0,0,0], [9E9, 9E9, 9E9, 9E9, 9E9, 9E9]];
	VAR robtarget Openhole_5708 := [[416.77, -24.13, 179.82], [-0.089611, 0.701406, 0.696153, 0.123979], [0,0,0,0], [9E9, 9E9, 9E9, 9E9, 9E9, 9E9]];
	VAR robtarget Openhole_5709 := [[416.27, -24.13, 179.8], [-0.091178, 0.701204, 0.695886, 0.125467], [0,0,0,0], [9E9, 9E9, 9E9, 9E9, 9E9, 9E9]];
	VAR robtarget Openhole_5710 := [[403.28, -23.96, 179.23], [-0.130623, 0.694937, 0.68832, 0.161914], [0,0,0,0], [9E9, 9E9, 9E9, 9E9, 9E9, 9E9]];
	VAR robtarget Openhole_5711 := [[402.79, -23.96, 179.21], [-0.132044, 0.694669, 0.688, 0.163267], [0,0,0,0], [9E9, 9E9, 9E9, 9E9, 9E9, 9E9]];
	VAR robtarget Openhole_5712 := [[396.3, -24.14, 178.81], [-0.14953, 0.691116, 0.683608, 0.180776], [0,0,0,0], [9E9, 9E9, 9E9, 9E9, 9E9, 9E9]];
	VAR robtarget Openhole_5713 := [[395.31, -24.2, 178.73], [-0.152044, 0.690567, 0.682892, 0.183462], [0,0,0,0], [9E9, 9E9, 9E9, 9E9, 9E9, 9E9]];
	VAR robtarget Openhole_5714 := [[394.34, -24.22, 178.67], [-0.154574, 0.690005, 0.682219, 0.185951], [0,0,0,0], [9E9, 9E9, 9E9, 9E9, 9E9, 9E9]];
	VAR robtarget Openhole_5715 := [[389.34, -24.22, 178.42], [-0.167619, 0.686953, 0.678778, 0.198142], [0,0,0,0], [9E9, 9E9, 9E9, 9E9, 9E9, 9E9]];
	VAR robtarget Openhole_5716 := [[362.34, -24.22, 178.51], [-0.183051, 0.683002, 0.683002, 0.183051], [0,0,0,0], [9E9, 9E9, 9E9, 9E9, 9E9, 9E9]];
	VAR robtarget Openhole_5717 := [[362.33, -26.32, 177.29], [-0.183051, 0.683002, 0.683002, 0.183051], [0,0,0,0], [9E9, 9E9, 9E9, 9E9, 9E9, 9E9]];
	VAR robtarget Openhole_5718 := [[389.33, -26.32, 177.21], [-0.161596, 0.688394, 0.677019, 0.204072], [0,0,0,0], [9E9, 9E9, 9E9, 9E9, 9E9, 9E9]];
	VAR robtarget Openhole_5719 := [[394.33, -26.32, 177.56], [-0.1484, 0.691359, 0.680532, 0.192032], [0,0,0,0], [9E9, 9E9, 9E9, 9E9, 9E9, 9E9]];
	VAR robtarget Openhole_5720 := [[394.33, -26.32, 177.56], [-0.148417, 0.691355, 0.680528, 0.192047], [0,0,0,0], [9E9, 9E9, 9E9, 9E9, 9E9, 9E9]];
	VAR robtarget Openhole_5721 := [[394.83, -26.28, 177.61], [-0.147179, 0.69162, 0.680908, 0.190694], [0,0,0,0], [9E9, 9E9, 9E9, 9E9, 9E9, 9E9]];
	VAR robtarget Openhole_5722 := [[400.3, -26.08, 178.09], [-0.132636, 0.694556, 0.684805, 0.176188], [0,0,0,0], [9E9, 9E9, 9E9, 9E9, 9E9, 9E9]];
	VAR robtarget Openhole_5723 := [[401.3, -26.08, 178.16], [-0.129824, 0.695087, 0.685476, 0.173559], [0,0,0,0], [9E9, 9E9, 9E9, 9E9, 9E9, 9E9]];
	VAR robtarget Openhole_5724 := [[401.8, -26.08, 178.19], [-0.128401, 0.695351, 0.685808, 0.172244], [0,0,0,0], [9E9, 9E9, 9E9, 9E9, 9E9, 9E9]];
	VAR robtarget Openhole_5725 := [[416.77, -26.42, 179.1], [-0.082258, 0.702306, 0.69482, 0.131247], [0,0,0,0], [9E9, 9E9, 9E9, 9E9, 9E9, 9E9]];
	VAR robtarget Openhole_5726 := [[417.27, -26.42, 179.14], [-0.080686, 0.702488, 0.695099, 0.12976], [0,0,0,0], [9E9, 9E9, 9E9, 9E9, 9E9, 9E9]];
	VAR robtarget Openhole_5727 := [[422.25, -26.24, 179.54], [-0.06532, 0.704083, 0.697841, 0.114099], [0,0,0,0], [9E9, 9E9, 9E9, 9E9, 9E9, 9E9]];
	VAR robtarget Openhole_5728 := [[426.2, -25.8, 179.91], [-0.053868, 0.705052, 0.699954, 0.10032], [0,0,0,0], [9E9, 9E9, 9E9, 9E9, 9E9, 9E9]];
	VAR robtarget Openhole_5729 := [[426.69, -25.72, 179.96], [-0.052516, 0.705154, 0.700212, 0.098508], [0,0,0,0], [9E9, 9E9, 9E9, 9E9, 9E9, 9E9]];
	VAR robtarget Openhole_5730 := [[428.64, -25.31, 180.17], [-0.04742, 0.705515, 0.701228, 0.090988], [0,0,0,0], [9E9, 9E9, 9E9, 9E9, 9E9, 9E9]];
	VAR robtarget Openhole_5731 := [[431.04, -24.65, 180.43], [-0.041681, 0.705877, 0.702443, 0.081078], [0,0,0,0], [9E9, 9E9, 9E9, 9E9, 9E9, 9E9]];
	VAR robtarget Openhole_5732 := [[431.98, -24.33, 180.54], [-0.039601, 0.705997, 0.702906, 0.076963], [0,0,0,0], [9E9, 9E9, 9E9, 9E9, 9E9, 9E9]];
	VAR robtarget Openhole_5733 := [[432.44, -24.15, 180.59], [-0.038642, 0.70605, 0.703133, 0.074861], [0,0,0,0], [9E9, 9E9, 9E9, 9E9, 9E9, 9E9]];
	VAR robtarget Openhole_5734 := [[433.36, -23.77, 180.69], [-0.036851, 0.706146, 0.703575, 0.070586], [0,0,0,0], [9E9, 9E9, 9E9, 9E9, 9E9, 9E9]];
	VAR robtarget Openhole_5735 := [[434.26, -23.35, 180.79], [-0.035242, 0.706228, 0.703999, 0.066223], [0,0,0,0], [9E9, 9E9, 9E9, 9E9, 9E9, 9E9]];
	VAR robtarget Openhole_5736 := [[435.15, -22.9, 180.89], [-0.033773, 0.7063, 0.704401, 0.061794], [0,0,0,0], [9E9, 9E9, 9E9, 9E9, 9E9, 9E9]];
	VAR robtarget Openhole_5737 := [[436.02, -22.42, 180.99], [-0.032458, 0.706361, 0.704781, 0.0573], [0,0,0,0], [9E9, 9E9, 9E9, 9E9, 9E9, 9E9]];
	VAR robtarget Openhole_5738 := [[436.45, -22.16, 181.03], [-0.031859, 0.706389, 0.704962, 0.055031], [0,0,0,0], [9E9, 9E9, 9E9, 9E9, 9E9, 9E9]];
	VAR robtarget Openhole_5739 := [[438.54, -20.81, 181.24], [-0.02937, 0.706497, 0.705767, 0.043508], [0,0,0,0], [9E9, 9E9, 9E9, 9E9, 9E9, 9E9]];
	VAR robtarget Openhole_5740 := [[438.97, -20.55, 181.27], [-0.028798, 0.70652, 0.705905, 0.041209], [0,0,0,0], [9E9, 9E9, 9E9, 9E9, 9E9, 9E9]];
	VAR robtarget Openhole_5741 := [[439.41, -20.32, 181.3], [-0.028096, 0.706548, 0.706034, 0.038942], [0,0,0,0], [9E9, 9E9, 9E9, 9E9, 9E9, 9E9]];
	VAR robtarget Openhole_5742 := [[439.86, -20.1, 181.32], [-0.027321, 0.706579, 0.706154, 0.036696], [0,0,0,0], [9E9, 9E9, 9E9, 9E9, 9E9, 9E9]];
	VAR robtarget Openhole_5743 := [[440.32, -19.89, 181.35], [-0.026498, 0.70661, 0.706266, 0.034464], [0,0,0,0], [9E9, 9E9, 9E9, 9E9, 9E9, 9E9]];
	VAR robtarget Openhole_5744 := [[440.77, -19.7, 181.37], [-0.025617, 0.706643, 0.706371, 0.032251], [0,0,0,0], [9E9, 9E9, 9E9, 9E9, 9E9, 9E9]];
	VAR robtarget Openhole_5745 := [[441.39, -19.52, 181.38], [-0.024125, 0.706695, 0.706487, 0.029593], [0,0,0,0], [9E9, 9E9, 9E9, 9E9, 9E9, 9E9]];
	VAR robtarget Openhole_5746 := [[443.53, -19.52, 181.39], [-0.016854, 0.706906, 0.706753, 0.022361], [0,0,0,0], [9E9, 9E9, 9E9, 9E9, 9E9, 9E9]];
	VAR robtarget Openhole_5747 := [[443.72, -20.63, 181.33], [-0.012413, 0.706998, 0.706648, 0.025468], [0,0,0,0], [9E9, 9E9, 9E9, 9E9, 9E9, 9E9]];
	VAR robtarget Openhole_5748 := [[441.58, -20.63, 181.3], [-0.019692, 0.706833, 0.70635, 0.032696], [0,0,0,0], [9E9, 9E9, 9E9, 9E9, 9E9, 9E9]];
	VAR robtarget Openhole_5749 := [[440.79, -20.96, 181.26], [-0.021259, 0.706787, 0.706166, 0.036472], [0,0,0,0], [9E9, 9E9, 9E9, 9E9, 9E9, 9E9]];
	VAR robtarget Openhole_5750 := [[438.24, -22.52, 181.05], [-0.024615, 0.706678, 0.705317, 0.050283], [0,0,0,0], [9E9, 9E9, 9E9, 9E9, 9E9, 9E9]];
	VAR robtarget Openhole_5751 := [[436.52, -23.52, 180.87], [-0.027047, 0.706589, 0.70461, 0.05937], [0,0,0,0], [9E9, 9E9, 9E9, 9E9, 9E9, 9E9]];
	VAR robtarget Openhole_5752 := [[435.19, -24.2, 180.72], [-0.029237, 0.706502, 0.704017, 0.066035], [0,0,0,0], [9E9, 9E9, 9E9, 9E9, 9E9, 9E9]];
	VAR robtarget Openhole_5753 := [[434.29, -24.62, 180.61], [-0.030863, 0.706433, 0.703594, 0.070399], [0,0,0,0], [9E9, 9E9, 9E9, 9E9, 9E9, 9E9]];
	VAR robtarget Openhole_5754 := [[433.83, -24.82, 180.56], [-0.031734, 0.706394, 0.703375, 0.072553], [0,0,0,0], [9E9, 9E9, 9E9, 9E9, 9E9, 9E9]];
	VAR robtarget Openhole_5755 := [[433.37, -25.01, 180.5], [-0.032645, 0.706353, 0.703152, 0.074686], [0,0,0,0], [9E9, 9E9, 9E9, 9E9, 9E9, 9E9]];
	VAR robtarget Openhole_5756 := [[432.91, -25.19, 180.45], [-0.033602, 0.706308, 0.702924, 0.076794], [0,0,0,0], [9E9, 9E9, 9E9, 9E9, 9E9, 9E9]];
	VAR robtarget Openhole_5757 := [[429.59, -26.22, 180.05], [-0.041252, 0.705902, 0.701234, 0.090944], [0,0,0,0], [9E9, 9E9, 9E9, 9E9, 9E9, 9E9]];
	VAR robtarget Openhole_5758 := [[426.18, -26.93, 179.66], [-0.050192, 0.705323, 0.699407, 0.104068], [0,0,0,0], [9E9, 9E9, 9E9, 9E9, 9E9, 9E9]];
	VAR robtarget Openhole_5759 := [[422.23, -27.36, 179.25], [-0.061718, 0.704408, 0.697234, 0.11775], [0,0,0,0], [9E9, 9E9, 9E9, 9E9, 9E9, 9E9]];
	VAR robtarget Openhole_5760 := [[416.76, -27.54, 178.75], [-0.078697, 0.702714, 0.694135, 0.134819], [0,0,0,0], [9E9, 9E9, 9E9, 9E9, 9E9, 9E9]];
	VAR robtarget Openhole_5761 := [[416.26, -27.54, 178.71], [-0.080278, 0.702535, 0.693849, 0.136284], [0,0,0,0], [9E9, 9E9, 9E9, 9E9, 9E9, 9E9]];
	VAR robtarget Openhole_5762 := [[405.79, -27.19, 178], [-0.1134, 0.697954, 0.687612, 0.164892], [0,0,0,0], [9E9, 9E9, 9E9, 9E9, 9E9, 9E9]];
	VAR robtarget Openhole_5763 := [[399.81, -27.04, 177.6], [-0.131167, 0.694835, 0.683732, 0.180306], [0,0,0,0], [9E9, 9E9, 9E9, 9E9, 9E9, 9E9]];
	VAR robtarget Openhole_5764 := [[399.31, -27.04, 177.56], [-0.132568, 0.694569, 0.683391, 0.181595], [0,0,0,0], [9E9, 9E9, 9E9, 9E9, 9E9, 9E9]];
	VAR robtarget Openhole_5765 := [[394.26, -27.21, 177.09], [-0.146024, 0.691865, 0.679758, 0.194755], [0,0,0,0], [9E9, 9E9, 9E9, 9E9, 9E9, 9E9]];
	VAR robtarget Openhole_5766 := [[389.33, -27.21, 176.7], [-0.159074, 0.688981, 0.676268, 0.206546], [0,0,0,0], [9E9, 9E9, 9E9, 9E9, 9E9, 9E9]];
	VAR robtarget Openhole_5767 := [[362.33, -27.21, 176.78], [-0.183051, 0.683002, 0.683002, 0.183051], [0,0,0,0], [9E9, 9E9, 9E9, 9E9, 9E9, 9E9]];
	VAR robtarget Openhole_5768 := [[362.33, -28.09, 176.27], [-0.183051, 0.683002, 0.683002, 0.183051], [0,0,0,0], [9E9, 9E9, 9E9, 9E9, 9E9, 9E9]];
	VAR robtarget Openhole_5769 := [[389.33, -28.09, 176.19], [-0.156549, 0.68956, 0.675508, 0.209019], [0,0,0,0], [9E9, 9E9, 9E9, 9E9, 9E9, 9E9]];
	VAR robtarget Openhole_5770 := [[394.33, -28.09, 176.62], [-0.143227, 0.692449, 0.67908, 0.197107], [0,0,0,0], [9E9, 9E9, 9E9, 9E9, 9E9, 9E9]];
	VAR robtarget Openhole_5771 := [[395.18, -28.08, 176.7], [-0.140929, 0.692921, 0.679681, 0.195022], [0,0,0,0], [9E9, 9E9, 9E9, 9E9, 9E9, 9E9]];
	VAR robtarget Openhole_5772 := [[398.16, -28.02, 176.99], [-0.132852, 0.694515, 0.681827, 0.187383], [0,0,0,0], [9E9, 9E9, 9E9, 9E9, 9E9, 9E9]];
	VAR robtarget Openhole_5773 := [[398.66, -28.02, 177.03], [-0.131447, 0.694782, 0.682171, 0.186124], [0,0,0,0], [9E9, 9E9, 9E9, 9E9, 9E9, 9E9]];
	VAR robtarget Openhole_5774 := [[405.64, -28.29, 177.53], [-0.110472, 0.698424, 0.686709, 0.168615], [0,0,0,0], [9E9, 9E9, 9E9, 9E9, 9E9, 9E9]];
	VAR robtarget Openhole_5775 := [[415.1, -28.72, 178.23], [-0.080132, 0.702552, 0.692412, 0.143406], [0,0,0,0], [9E9, 9E9, 9E9, 9E9, 9E9, 9E9]];
	VAR robtarget Openhole_5776 := [[417.09, -28.75, 178.4], [-0.073749, 0.70325, 0.693581, 0.137645], [0,0,0,0], [9E9, 9E9, 9E9, 9E9, 9E9, 9E9]];
	VAR robtarget Openhole_5777 := [[417.59, -28.74, 178.45], [-0.072169, 0.703414, 0.693872, 0.136167], [0,0,0,0], [9E9, 9E9, 9E9, 9E9, 9E9, 9E9]];
	VAR robtarget Openhole_5778 := [[423.06, -28.53, 179.02], [-0.0552, 0.704949, 0.697023, 0.118989], [0,0,0,0], [9E9, 9E9, 9E9, 9E9, 9E9, 9E9]];
	VAR robtarget Openhole_5779 := [[427, -28.06, 179.48], [-0.043757, 0.705752, 0.699238, 0.105193], [0,0,0,0], [9E9, 9E9, 9E9, 9E9, 9E9, 9E9]];
	VAR robtarget Openhole_5780 := [[430.4, -27.35, 179.9], [-0.034786, 0.706251, 0.701089, 0.092057], [0,0,0,0], [9E9, 9E9, 9E9, 9E9, 9E9, 9E9]];
	VAR robtarget Openhole_5781 := [[432.32, -26.83, 180.14], [-0.030104, 0.706466, 0.702081, 0.084155], [0,0,0,0], [9E9, 9E9, 9E9, 9E9, 9E9, 9E9]];
	VAR robtarget Openhole_5782 := [[433.73, -26.37, 180.32], [-0.026858, 0.706597, 0.702788, 0.078031], [0,0,0,0], [9E9, 9E9, 9E9, 9E9, 9E9, 9E9]];
	VAR robtarget Openhole_5783 := [[434.67, -26.03, 180.43], [-0.024862, 0.70667, 0.70324, 0.073843], [0,0,0,0], [9E9, 9E9, 9E9, 9E9, 9E9, 9E9]];
	VAR robtarget Openhole_5784 := [[437.86, -24.65, 180.8], [-0.018706, 0.706859, 0.704667, 0.058688], [0,0,0,0], [9E9, 9E9, 9E9, 9E9, 9E9, 9E9]];
	VAR robtarget Openhole_5785 := [[438.31, -24.43, 180.85], [-0.017944, 0.706879, 0.704849, 0.056462], [0,0,0,0], [9E9, 9E9, 9E9, 9E9, 9E9, 9E9]];
	VAR robtarget Openhole_5786 := [[439.62, -23.72, 180.98], [-0.015871, 0.706929, 0.705358, 0.049696], [0,0,0,0], [9E9, 9E9, 9E9, 9E9, 9E9, 9E9]];
	VAR robtarget Openhole_5787 := [[440.05, -23.46, 181.02], [-0.015286, 0.706942, 0.705516, 0.047405], [0,0,0,0], [9E9, 9E9, 9E9, 9E9, 9E9, 9E9]];
	VAR robtarget Openhole_5788 := [[441.31, -22.66, 181.14], [-0.013721, 0.706974, 0.705948, 0.040466], [0,0,0,0], [9E9, 9E9, 9E9, 9E9, 9E9, 9E9]];
	VAR robtarget Openhole_5789 := [[442.15, -22.2, 181.2], [-0.012426, 0.706998, 0.706186, 0.036084], [0,0,0,0], [9E9, 9E9, 9E9, 9E9, 9E9, 9E9]];
	VAR robtarget Openhole_5790 := [[443.96, -22.2, 181.26], [-0.006283, 0.707079, 0.70647, 0.029995], [0,0,0,0], [9E9, 9E9, 9E9, 9E9, 9E9, 9E9]];
	VAR robtarget Openhole_5791 := [[445.39, -24.26, 181.22], [0.0056, 0.707085, 0.706378, 0.032093], [0,0,0,0], [9E9, 9E9, 9E9, 9E9, 9E9, 9E9]];
	VAR robtarget Openhole_5792 := [[443.59, -24.26, 181.13], [-0.000555, 0.707107, 0.706075, 0.038187], [0,0,0,0], [9E9, 9E9, 9E9, 9E9, 9E9, 9E9]];
	VAR robtarget Openhole_5793 := [[442.83, -24.81, 181.06], [-0.00127, 0.707106, 0.705822, 0.04261], [0,0,0,0], [9E9, 9E9, 9E9, 9E9, 9E9, 9E9]];
	VAR robtarget Openhole_5794 := [[441.94, -25.27, 180.98], [-0.002739, 0.707101, 0.705535, 0.047127], [0,0,0,0], [9E9, 9E9, 9E9, 9E9, 9E9, 9E9]];
	VAR robtarget Openhole_5795 := [[441.49, -25.47, 180.93], [-0.003612, 0.707098, 0.705384, 0.049332], [0,0,0,0], [9E9, 9E9, 9E9, 9E9, 9E9, 9E9]];
	VAR robtarget Openhole_5796 := [[441.02, -25.65, 180.89], [-0.004591, 0.707092, 0.70523, 0.051491], [0,0,0,0], [9E9, 9E9, 9E9, 9E9, 9E9, 9E9]];
	VAR robtarget Openhole_5797 := [[439.61, -26.14, 180.76], [-0.007707, 0.707065, 0.704735, 0.057865], [0,0,0,0], [9E9, 9E9, 9E9, 9E9, 9E9, 9E9]];
	VAR robtarget Openhole_5798 := [[433.43, -28.02, 180.04], [-0.022341, 0.706754, 0.702042, 0.084483], [0,0,0,0], [9E9, 9E9, 9E9, 9E9, 9E9, 9E9]];
	VAR robtarget Openhole_5799 := [[429.08, -29, 179.48], [-0.033733, 0.706302, 0.699757, 0.101684], [0,0,0,0], [9E9, 9E9, 9E9, 9E9, 9E9, 9E9]];
	VAR robtarget Openhole_5800 := [[424.66, -29.62, 178.9], [-0.046355, 0.705586, 0.697266, 0.117562], [0,0,0,0], [9E9, 9E9, 9E9, 9E9, 9E9, 9E9]];
	VAR robtarget Openhole_5801 := [[420.2, -29.9, 178.37], [-0.060029, 0.704554, 0.694668, 0.132049], [0,0,0,0], [9E9, 9E9, 9E9, 9E9, 9E9, 9E9]];
	VAR robtarget Openhole_5802 := [[417.72, -29.94, 178.1], [-0.067913, 0.703838, 0.693196, 0.13957], [0,0,0,0], [9E9, 9E9, 9E9, 9E9, 9E9, 9E9]];
	VAR robtarget Openhole_5803 := [[417.22, -29.94, 178.05], [-0.069512, 0.703682, 0.6929, 0.141028], [0,0,0,0], [9E9, 9E9, 9E9, 9E9, 9E9, 9E9]];
	VAR robtarget Openhole_5804 := [[410.75, -29.69, 177.46], [-0.090619, 0.701276, 0.689039, 0.158826], [0,0,0,0], [9E9, 9E9, 9E9, 9E9, 9E9, 9E9]];
	VAR robtarget Openhole_5805 := [[399.3, -28.99, 176.63], [-0.126733, 0.695657, 0.681847, 0.18731], [0,0,0,0], [9E9, 9E9, 9E9, 9E9, 9E9, 9E9]];
	VAR robtarget Openhole_5806 := [[396.81, -28.94, 176.41], [-0.133871, 0.694319, 0.680131, 0.193446], [0,0,0,0], [9E9, 9E9, 9E9, 9E9, 9E9, 9E9]];
	VAR robtarget Openhole_5807 := [[396.32, -28.94, 176.36], [-0.135249, 0.694052, 0.679777, 0.194686], [0,0,0,0], [9E9, 9E9, 9E9, 9E9, 9E9, 9E9]];
	VAR robtarget Openhole_5808 := [[394.83, -28.97, 176.21], [-0.139297, 0.693251, 0.678697, 0.198418], [0,0,0,0], [9E9, 9E9, 9E9, 9E9, 9E9, 9E9]];
	VAR robtarget Openhole_5809 := [[394.3, -28.99, 176.14], [-0.140653, 0.692977, 0.678305, 0.199754], [0,0,0,0], [9E9, 9E9, 9E9, 9E9, 9E9, 9E9]];
	VAR robtarget Openhole_5810 := [[389.33, -28.99, 175.67], [-0.153969, 0.69014, 0.674722, 0.211542], [0,0,0,0], [9E9, 9E9, 9E9, 9E9, 9E9, 9E9]];
	VAR robtarget Openhole_5811 := [[362.33, -28.99, 175.75], [-0.183051, 0.683002, 0.683002, 0.183051], [0,0,0,0], [9E9, 9E9, 9E9, 9E9, 9E9, 9E9]];
	VAR robtarget Openhole_5812 := [[362.33, -30.66, 174.79], [-0.183051, 0.683002, 0.683002, 0.183051], [0,0,0,0], [9E9, 9E9, 9E9, 9E9, 9E9, 9E9]];
	VAR robtarget Openhole_5813 := [[374.33, -30.66, 174.75], [-0.183051, 0.683002, 0.683002, 0.183051], [0,0,0,0], [9E9, 9E9, 9E9, 9E9, 9E9, 9E9]];
	VAR robtarget Openhole_5814 := [[389.33, -30.66, 174.7], [-0.149199, 0.691187, 0.673247, 0.216191], [0,0,0,0], [9E9, 9E9, 9E9, 9E9, 9E9, 9E9]];
	VAR robtarget Openhole_5815 := [[394.83, -30.66, 175.32], [-0.134293, 0.694237, 0.677263, 0.203261], [0,0,0,0], [9E9, 9E9, 9E9, 9E9, 9E9, 9E9]];
	VAR robtarget Openhole_5816 := [[399.31, -30.93, 175.69], [-0.12089, 0.696696, 0.68026, 0.192993], [0,0,0,0], [9E9, 9E9, 9E9, 9E9, 9E9, 9E9]];
	VAR robtarget Openhole_5817 := [[410.71, -32.09, 176.56], [-0.083207, 0.702194, 0.687276, 0.166289], [0,0,0,0], [9E9, 9E9, 9E9, 9E9, 9E9, 9E9]];
	VAR robtarget Openhole_5818 := [[417.16, -32.5, 177.25], [-0.061502, 0.704427, 0.691185, 0.14921], [0,0,0,0], [9E9, 9E9, 9E9, 9E9, 9E9, 9E9]];
	VAR robtarget Openhole_5819 := [[419.64, -32.54, 177.56], [-0.053332, 0.705093, 0.692691, 0.142055], [0,0,0,0], [9E9, 9E9, 9E9, 9E9, 9E9, 9E9]];
	VAR robtarget Openhole_5820 := [[420.14, -32.54, 177.62], [-0.051716, 0.705213, 0.692991, 0.140582], [0,0,0,0], [9E9, 9E9, 9E9, 9E9, 9E9, 9E9]];
	VAR robtarget Openhole_5821 := [[425.09, -32.35, 178.31], [-0.036014, 0.706189, 0.695968, 0.125016], [0,0,0,0], [9E9, 9E9, 9E9, 9E9, 9E9, 9E9]];
	VAR robtarget Openhole_5822 := [[430.5, -31.78, 179.11], [-0.019738, 0.706831, 0.699077, 0.106263], [0,0,0,0], [9E9, 9E9, 9E9, 9E9, 9E9, 9E9]];
	VAR robtarget Openhole_5823 := [[437.38, -30.92, 180.05], [0.000755, 0.707106, 0.702431, 0.081185], [0,0,0,0], [9E9, 9E9, 9E9, 9E9, 9E9, 9E9]];
	VAR robtarget Openhole_5824 := [[438.37, -30.84, 180.17], [0.003846, 0.707096, 0.70283, 0.077652], [0,0,0,0], [9E9, 9E9, 9E9, 9E9, 9E9, 9E9]];
	VAR robtarget Openhole_5825 := [[439.36, -30.78, 180.29], [0.007039, 0.707072, 0.703204, 0.074188], [0,0,0,0], [9E9, 9E9, 9E9, 9E9, 9E9, 9E9]];
	VAR robtarget Openhole_5826 := [[440.85, -30.75, 180.46], [0.012008, 0.707005, 0.70372, 0.069128], [0,0,0,0], [9E9, 9E9, 9E9, 9E9, 9E9, 9E9]];
	VAR robtarget Openhole_5827 := [[441.35, -30.75, 180.52], [0.013708, 0.706974, 0.70388, 0.067476], [0,0,0,0], [9E9, 9E9, 9E9, 9E9, 9E9, 9E9]];
	VAR robtarget Openhole_5828 := [[445.32, -30.96, 180.96], [0.027984, 0.706553, 0.704973, 0.05489], [0,0,0,0], [9E9, 9E9, 9E9, 9E9, 9E9, 9E9]];
	VAR robtarget Openhole_5829 := [[449.27, -31.31, 181.41], [0.042673, 0.705818, 0.705816, 0.042711], [0,0,0,0], [9E9, 9E9, 9E9, 9E9, 9E9, 9E9]];
	VAR robtarget Openhole_5830 := [[449.77, -31.34, 181.47], [0.044436, 0.705709, 0.705911, 0.041104], [0,0,0,0], [9E9, 9E9, 9E9, 9E9, 9E9, 9E9]];
	VAR robtarget Openhole_5831 := [[450.27, -31.35, 181.53], [0.04617, 0.705598, 0.706005, 0.039466], [0,0,0,0], [9E9, 9E9, 9E9, 9E9, 9E9, 9E9]];
	VAR robtarget Openhole_5832 := [[450.76, -31.35, 181.59], [0.047855, 0.705486, 0.706097, 0.037782], [0,0,0,0], [9E9, 9E9, 9E9, 9E9, 9E9, 9E9]];
	VAR robtarget Openhole_5833 := [[451.76, -31.32, 181.71], [0.051098, 0.705258, 0.706275, 0.034288], [0,0,0,0], [9E9, 9E9, 9E9, 9E9, 9E9, 9E9]];
	VAR robtarget Openhole_5834 := [[452.75, -31.23, 181.82], [0.054163, 0.705029, 0.706443, 0.030638], [0,0,0,0], [9E9, 9E9, 9E9, 9E9, 9E9, 9E9]];
	VAR robtarget Openhole_5835 := [[453.73, -31.11, 181.93], [0.057088, 0.704799, 0.706596, 0.026875], [0,0,0,0], [9E9, 9E9, 9E9, 9E9, 9E9, 9E9]];
	VAR robtarget Openhole_5836 := [[461.6, -29.87, 182.7], [0.079204, 0.702657, 0.707095, -0.004031], [0,0,0,0], [9E9, 9E9, 9E9, 9E9, 9E9, 9E9]];
	VAR robtarget Openhole_5837 := [[470.53, -29.03, 183.46], [0.105282, 0.699225, 0.706145, -0.036867], [0,0,0,0], [9E9, 9E9, 9E9, 9E9, 9E9, 9E9]];
	VAR robtarget Openhole_5838 := [[482.96, -28.21, 184.39], [0.140615, 0.692984, 0.702583, -0.079861], [0,0,0,0], [9E9, 9E9, 9E9, 9E9, 9E9, 9E9]];
	VAR robtarget Openhole_5839 := [[502.4, -27.36, 185.68], [0.19086, 0.680862, 0.693126, -0.139915], [0,0,0,0], [9E9, 9E9, 9E9, 9E9, 9E9, 9E9]];
	VAR robtarget Openhole_5840 := [[504.36, -27.26, 185.78], [0.195417, 0.679568, 0.691965, -0.145547], [0,0,0,0], [9E9, 9E9, 9E9, 9E9, 9E9, 9E9]];
	VAR robtarget Openhole_5841 := [[509.36, -27.26, 186.18], [0.183051, 0.683002, 0.683002, -0.183051], [0,0,0,0], [9E9, 9E9, 9E9, 9E9, 9E9, 9E9]];
	VAR robtarget Openhole_5842 := [[536.36, -27.26, 186.09], [0.183051, 0.683002, 0.683002, -0.183051], [0,0,0,0], [9E9, 9E9, 9E9, 9E9, 9E9, 9E9]];
	VAR robtarget Openhole_5843 := [[536.36, -28.38, 186.74], [0.183051, 0.683002, 0.683002, -0.183051], [0,0,0,0], [9E9, 9E9, 9E9, 9E9, 9E9, 9E9]];
	VAR robtarget Openhole_5844 := [[509.36, -28.38, 186.83], [0.183051, 0.683002, 0.683002, -0.183051], [0,0,0,0], [9E9, 9E9, 9E9, 9E9, 9E9, 9E9]];
	VAR robtarget Openhole_5845 := [[504.36, -28.38, 186.38], [0.198634, 0.678634, 0.692645, -0.142276], [0,0,0,0], [9E9, 9E9, 9E9, 9E9, 9E9, 9E9]];
	VAR robtarget Openhole_5846 := [[483.57, -29.45, 184.85], [0.146274, 0.691812, 0.702813, -0.077803], [0,0,0,0], [9E9, 9E9, 9E9, 9E9, 9E9, 9E9]];
	VAR robtarget Openhole_5847 := [[473.63, -30.27, 184.05], [0.119031, 0.697016, 0.705792, -0.043103], [0,0,0,0], [9E9, 9E9, 9E9, 9E9, 9E9, 9E9]];
	VAR robtarget Openhole_5848 := [[466.22, -31.16, 183.39], [0.098507, 0.700212, 0.706939, -0.015381], [0,0,0,0], [9E9, 9E9, 9E9, 9E9, 9E9, 9E9]];
	VAR robtarget Openhole_5849 := [[460.33, -32.16, 182.81], [0.082599, 0.702266, 0.707063, 0.007897], [0,0,0,0], [9E9, 9E9, 9E9, 9E9, 9E9, 9E9]];
	VAR robtarget Openhole_5850 := [[452.59, -33.96, 181.89], [0.062751, 0.704317, 0.705959, 0.040273], [0,0,0,0], [9E9, 9E9, 9E9, 9E9, 9E9, 9E9]];
	VAR robtarget Openhole_5851 := [[452.1, -34.05, 181.82], [0.061375, 0.704438, 0.705846, 0.042207], [0,0,0,0], [9E9, 9E9, 9E9, 9E9, 9E9, 9E9]];
	VAR robtarget Openhole_5852 := [[451.61, -34.11, 181.75], [0.059939, 0.704562, 0.70573, 0.044098], [0,0,0,0], [9E9, 9E9, 9E9, 9E9, 9E9, 9E9]];
	VAR robtarget Openhole_5853 := [[451.12, -34.17, 181.68], [0.058451, 0.704687, 0.705612, 0.045946], [0,0,0,0], [9E9, 9E9, 9E9, 9E9, 9E9, 9E9]];
	VAR robtarget Openhole_5854 := [[450.63, -34.2, 181.61], [0.056888, 0.704815, 0.705494, 0.047732], [0,0,0,0], [9E9, 9E9, 9E9, 9E9, 9E9, 9E9]];
	VAR robtarget Openhole_5855 := [[450.13, -34.22, 181.54], [0.055276, 0.704943, 0.705374, 0.049473], [0,0,0,0], [9E9, 9E9, 9E9, 9E9, 9E9, 9E9]];
	VAR robtarget Openhole_5856 := [[449.64, -34.22, 181.46], [0.053595, 0.705073, 0.705254, 0.051149], [0,0,0,0], [9E9, 9E9, 9E9, 9E9, 9E9, 9E9]];
	VAR robtarget Openhole_5857 := [[449.14, -34.2, 181.39], [0.051869, 0.705202, 0.705134, 0.052778], [0,0,0,0], [9E9, 9E9, 9E9, 9E9, 9E9, 9E9]];
	VAR robtarget Openhole_5858 := [[448.65, -34.17, 181.32], [0.050076, 0.705331, 0.705016, 0.054336], [0,0,0,0], [9E9, 9E9, 9E9, 9E9, 9E9, 9E9]];
	VAR robtarget Openhole_5859 := [[448.16, -34.12, 181.25], [0.048239, 0.705459, 0.704899, 0.05584], [0,0,0,0], [9E9, 9E9, 9E9, 9E9, 9E9, 9E9]];
	VAR robtarget Openhole_5860 := [[447.66, -34.06, 181.18], [0.04636, 0.705585, 0.704782, 0.057294], [0,0,0,0], [9E9, 9E9, 9E9, 9E9, 9E9, 9E9]];
	VAR robtarget Openhole_5861 := [[442.77, -33.27, 180.52], [0.027009, 0.706591, 0.703524, 0.071091], [0,0,0,0], [9E9, 9E9, 9E9, 9E9, 9E9, 9E9]];
	VAR robtarget Openhole_5862 := [[439.31, -33.03, 180.07], [0.01437, 0.706961, 0.702361, 0.081787], [0,0,0,0], [9E9, 9E9, 9E9, 9E9, 9E9, 9E9]];
	VAR robtarget Openhole_5863 := [[438.32, -33.02, 179.94], [0.010944, 0.707022, 0.701978, 0.085012], [0,0,0,0], [9E9, 9E9, 9E9, 9E9, 9E9, 9E9]];
	VAR robtarget Openhole_5864 := [[437.82, -33.02, 179.87], [0.00927, 0.707046, 0.701777, 0.086658], [0,0,0,0], [9E9, 9E9, 9E9, 9E9, 9E9, 9E9]];
	VAR robtarget Openhole_5865 := [[433.38, -33.3, 179.23], [-0.004982, 0.707089, 0.699714, 0.101983], [0,0,0,0], [9E9, 9E9, 9E9, 9E9, 9E9, 9E9]];
	VAR robtarget Openhole_5866 := [[425.51, -33.98, 177.99], [-0.029319, 0.706499, 0.695253, 0.128929], [0,0,0,0], [9E9, 9E9, 9E9, 9E9, 9E9, 9E9]];
	VAR robtarget Openhole_5867 := [[421.06, -34.1, 177.32], [-0.043682, 0.705756, 0.692546, 0.142758], [0,0,0,0], [9E9, 9E9, 9E9, 9E9, 9E9, 9E9]];
	VAR robtarget Openhole_5868 := [[420.56, -34.09, 177.25], [-0.045314, 0.705653, 0.692242, 0.144224], [0,0,0,0], [9E9, 9E9, 9E9, 9E9, 9E9, 9E9]];
	VAR robtarget Openhole_5869 := [[415.12, -33.89, 176.53], [-0.063661, 0.704235, 0.688902, 0.159417], [0,0,0,0], [9E9, 9E9, 9E9, 9E9, 9E9, 9E9]];
	VAR robtarget Openhole_5870 := [[408.68, -33.3, 175.84], [-0.085753, 0.701888, 0.68498, 0.175506], [0,0,0,0], [9E9, 9E9, 9E9, 9E9, 9E9, 9E9]];
	VAR robtarget Openhole_5871 := [[400.77, -32.26, 175.24], [-0.112666, 0.698073, 0.680212, 0.193162], [0,0,0,0], [9E9, 9E9, 9E9, 9E9, 9E9, 9E9]];
	VAR robtarget Openhole_5872 := [[395.82, -31.65, 174.92], [-0.128628, 0.695309, 0.677133, 0.203692], [0,0,0,0], [9E9, 9E9, 9E9, 9E9, 9E9, 9E9]];
	VAR robtarget Openhole_5873 := [[394.83, -31.57, 174.84], [-0.131638, 0.694746, 0.676477, 0.20586], [0,0,0,0], [9E9, 9E9, 9E9, 9E9, 9E9, 9E9]];
	VAR robtarget Openhole_5874 := [[394.33, -31.54, 174.8], [-0.133102, 0.694467, 0.676139, 0.206968], [0,0,0,0], [9E9, 9E9, 9E9, 9E9, 9E9, 9E9]];
	VAR robtarget Openhole_5875 := [[389.32, -31.54, 174.19], [-0.146676, 0.691727, 0.672455, 0.218643], [0,0,0,0], [9E9, 9E9, 9E9, 9E9, 9E9, 9E9]];
	VAR robtarget Openhole_5876 := [[362.32, -31.54, 174.28], [-0.183051, 0.683002, 0.683002, 0.183051], [0,0,0,0], [9E9, 9E9, 9E9, 9E9, 9E9, 9E9]];
	VAR robtarget Openhole_5877 := [[362.32, -32.55, 173.7], [-0.183051, 0.683002, 0.683002, 0.183051], [0,0,0,0], [9E9, 9E9, 9E9, 9E9, 9E9, 9E9]];
	VAR robtarget Openhole_5878 := [[389.32, -32.55, 173.61], [-0.143805, 0.692329, 0.671543, 0.221427], [0,0,0,0], [9E9, 9E9, 9E9, 9E9, 9E9, 9E9]];
	VAR robtarget Openhole_5879 := [[394.32, -32.55, 174.26], [-0.130172, 0.695022, 0.675256, 0.209831], [0,0,0,0], [9E9, 9E9, 9E9, 9E9, 9E9, 9E9]];
	VAR robtarget Openhole_5880 := [[395.25, -32.64, 174.34], [-0.127334, 0.695547, 0.675858, 0.207883], [0,0,0,0], [9E9, 9E9, 9E9, 9E9, 9E9, 9E9]];
	VAR robtarget Openhole_5881 := [[405.09, -34.29, 174.92], [-0.093678, 0.700874, 0.681654, 0.188008], [0,0,0,0], [9E9, 9E9, 9E9, 9E9, 9E9, 9E9]];
	VAR robtarget Openhole_5882 := [[411.51, -35.11, 175.57], [-0.071294, 0.703503, 0.685549, 0.173268], [0,0,0,0], [9E9, 9E9, 9E9, 9E9, 9E9, 9E9]];
	VAR robtarget Openhole_5883 := [[417.44, -35.57, 176.34], [-0.050831, 0.705277, 0.689238, 0.15796], [0,0,0,0], [9E9, 9E9, 9E9, 9E9, 9E9, 9E9]];
	VAR robtarget Openhole_5884 := [[421.88, -35.68, 177.02], [-0.035866, 0.706197, 0.692023, 0.145274], [0,0,0,0], [9E9, 9E9, 9E9, 9E9, 9E9, 9E9]];
	VAR robtarget Openhole_5885 := [[422.38, -35.68, 177.1], [-0.034238, 0.706277, 0.692332, 0.143792], [0,0,0,0], [9E9, 9E9, 9E9, 9E9, 9E9, 9E9]];
	VAR robtarget Openhole_5886 := [[428.29, -35.44, 178.1], [-0.015208, 0.706943, 0.69597, 0.125003], [0,0,0,0], [9E9, 9E9, 9E9, 9E9, 9E9, 9E9]];
	VAR robtarget Openhole_5887 := [[436.16, -34.91, 179.41], [0.009849, 0.707038, 0.700245, 0.098267], [0,0,0,0], [9E9, 9E9, 9E9, 9E9, 9E9, 9E9]];
	VAR robtarget Openhole_5888 := [[437.15, -34.9, 179.56], [0.01318, 0.706984, 0.700696, 0.095004], [0,0,0,0], [9E9, 9E9, 9E9, 9E9, 9E9, 9E9]];
	VAR robtarget Openhole_5889 := [[437.64, -34.9, 179.63], [0.014872, 0.70695, 0.700912, 0.093394], [0,0,0,0], [9E9, 9E9, 9E9, 9E9, 9E9, 9E9]];
	VAR robtarget Openhole_5890 := [[439.13, -34.94, 179.86], [0.020087, 0.706821, 0.701525, 0.08867], [0,0,0,0], [9E9, 9E9, 9E9, 9E9, 9E9, 9E9]];
	VAR robtarget Openhole_5891 := [[440.11, -35, 180], [0.023684, 0.70671, 0.701902, 0.085633], [0,0,0,0], [9E9, 9E9, 9E9, 9E9, 9E9, 9E9]];
	VAR robtarget Openhole_5892 := [[443.55, -35.46, 180.5], [0.036964, 0.70614, 0.703036, 0.075764], [0,0,0,0], [9E9, 9E9, 9E9, 9E9, 9E9, 9E9]];
	VAR robtarget Openhole_5893 := [[446.93, -36.18, 181.02], [0.050888, 0.705273, 0.703949, 0.06675], [0,0,0,0], [9E9, 9E9, 9E9, 9E9, 9E9, 9E9]];
	VAR robtarget Openhole_5894 := [[447.42, -36.26, 181.1], [0.052826, 0.705131, 0.704077, 0.065392], [0,0,0,0], [9E9, 9E9, 9E9, 9E9, 9E9, 9E9]];
	VAR robtarget Openhole_5895 := [[447.91, -36.33, 181.18], [0.054732, 0.704985, 0.704205, 0.063989], [0,0,0,0], [9E9, 9E9, 9E9, 9E9, 9E9, 9E9]];
	VAR robtarget Openhole_5896 := [[448.4, -36.38, 181.26], [0.05656, 0.704841, 0.70434, 0.06249], [0,0,0,0], [9E9, 9E9, 9E9, 9E9, 9E9, 9E9]];
	VAR robtarget Openhole_5897 := [[448.89, -36.4, 181.35], [0.058287, 0.7047, 0.704482, 0.060874], [0,0,0,0], [9E9, 9E9, 9E9, 9E9, 9E9, 9E9]];
	VAR robtarget Openhole_5898 := [[449.38, -36.38, 181.43], [0.059912, 0.704564, 0.704628, 0.059157], [0,0,0,0], [9E9, 9E9, 9E9, 9E9, 9E9, 9E9]];
	VAR robtarget Openhole_5899 := [[449.87, -36.33, 181.51], [0.06141, 0.704435, 0.704779, 0.057331], [0,0,0,0], [9E9, 9E9, 9E9, 9E9, 9E9, 9E9]];
	VAR robtarget Openhole_5900 := [[450.85, -36.17, 181.67], [0.064158, 0.70419, 0.705081, 0.053484], [0,0,0,0], [9E9, 9E9, 9E9, 9E9, 9E9, 9E9]];
	VAR robtarget Openhole_5901 := [[455.16, -35.07, 182.32], [0.075046, 0.703113, 0.706232, 0.035169], [0,0,0,0], [9E9, 9E9, 9E9, 9E9, 9E9, 9E9]];
	VAR robtarget Openhole_5902 := [[460.92, -33.54, 183.04], [0.089087, 0.701472, 0.707029, 0.010462], [0,0,0,0], [9E9, 9E9, 9E9, 9E9, 9E9, 9E9]];
	VAR robtarget Openhole_5903 := [[466.77, -32.38, 183.66], [0.104279, 0.699375, 0.706983, -0.013234], [0,0,0,0], [9E9, 9E9, 9E9, 9E9, 9E9, 9E9]];
	VAR robtarget Openhole_5904 := [[473.67, -31.4, 184.32], [0.122798, 0.696363, 0.706001, -0.039535], [0,0,0,0], [9E9, 9E9, 9E9, 9E9, 9E9, 9E9]];
	VAR robtarget Openhole_5905 := [[482.1, -30.56, 185.06], [0.145477, 0.69198, 0.703672, -0.069607], [0,0,0,0], [9E9, 9E9, 9E9, 9E9, 9E9, 9E9]];
	VAR robtarget Openhole_5906 := [[494.53, -29.79, 186.1], [0.177766, 0.684397, 0.698469, -0.110186], [0,0,0,0], [9E9, 9E9, 9E9, 9E9, 9E9, 9E9]];
	VAR robtarget Openhole_5907 := [[504.36, -29.28, 186.85], [0.201187, 0.677882, 0.693174, -0.139675], [0,0,0,0], [9E9, 9E9, 9E9, 9E9, 9E9, 9E9]];
	VAR robtarget Openhole_5908 := [[509.37, -29.28, 187.34], [0.183051, 0.683002, 0.683002, -0.183051], [0,0,0,0], [9E9, 9E9, 9E9, 9E9, 9E9, 9E9]];
	VAR robtarget Openhole_5909 := [[536.37, -29.28, 187.26], [0.183051, 0.683002, 0.683002, -0.183051], [0,0,0,0], [9E9, 9E9, 9E9, 9E9, 9E9, 9E9]];
	VAR robtarget Openhole_5910 := [[536.37, -30.16, 187.77], [0.183051, 0.683002, 0.683002, -0.183051], [0,0,0,0], [9E9, 9E9, 9E9, 9E9, 9E9, 9E9]];
	VAR robtarget Openhole_5911 := [[524.37, -30.16, 187.8], [0.183051, 0.683002, 0.683002, -0.183051], [0,0,0,0], [9E9, 9E9, 9E9, 9E9, 9E9, 9E9]];
	VAR robtarget Openhole_5912 := [[509.37, -30.16, 187.85], [0.183051, 0.683002, 0.683002, -0.183051], [0,0,0,0], [9E9, 9E9, 9E9, 9E9, 9E9, 9E9]];
	VAR robtarget Openhole_5913 := [[504.38, -30.16, 187.32], [0.20374, 0.677119, 0.693682, -0.13713], [0,0,0,0], [9E9, 9E9, 9E9, 9E9, 9E9, 9E9]];
	VAR robtarget Openhole_5914 := [[485.97, -31.27, 185.74], [0.158826, 0.689039, 0.702615, -0.079574], [0,0,0,0], [9E9, 9E9, 9E9, 9E9, 9E9, 9E9]];
	VAR robtarget Openhole_5915 := [[477.54, -32.07, 184.96], [0.136736, 0.69376, 0.705331, -0.050083], [0,0,0,0], [9E9, 9E9, 9E9, 9E9, 9E9, 9E9]];
	VAR robtarget Openhole_5916 := [[470.15, -33.11, 184.24], [0.117374, 0.697297, 0.706758, -0.022201], [0,0,0,0], [9E9, 9E9, 9E9, 9E9, 9E9, 9E9]];
	VAR robtarget Openhole_5917 := [[463.32, -34.47, 183.5], [0.099985, 0.700002, 0.707087, 0.005338], [0,0,0,0], [9E9, 9E9, 9E9, 9E9, 9E9, 9E9]];
	VAR robtarget Openhole_5918 := [[457.09, -36.14, 182.7], [0.085021, 0.701977, 0.706377, 0.032115], [0,0,0,0], [9E9, 9E9, 9E9, 9E9, 9E9, 9E9]];
	VAR robtarget Openhole_5919 := [[450.91, -37.89, 181.71], [0.07006, 0.703627, 0.704647, 0.058929], [0,0,0,0], [9E9, 9E9, 9E9, 9E9, 9E9, 9E9]];
	VAR robtarget Openhole_5920 := [[449.96, -38.12, 181.53], [0.067561, 0.703872, 0.704302, 0.062919], [0,0,0,0], [9E9, 9E9, 9E9, 9E9, 9E9, 9E9]];
	VAR robtarget Openhole_5921 := [[449.47, -38.19, 181.44], [0.066128, 0.704008, 0.704133, 0.064785], [0,0,0,0], [9E9, 9E9, 9E9, 9E9, 9E9, 9E9]];
	VAR robtarget Openhole_5922 := [[448.98, -38.23, 181.35], [0.06461, 0.704149, 0.703965, 0.066586], [0,0,0,0], [9E9, 9E9, 9E9, 9E9, 9E9, 9E9]];
	VAR robtarget Openhole_5923 := [[448.49, -38.23, 181.26], [0.062935, 0.7043, 0.703806, 0.068242], [0,0,0,0], [9E9, 9E9, 9E9, 9E9, 9E9, 9E9]];
	VAR robtarget Openhole_5924 := [[448, -38.2, 181.17], [0.061187, 0.704454, 0.703651, 0.06982], [0,0,0,0], [9E9, 9E9, 9E9, 9E9, 9E9, 9E9]];
	VAR robtarget Openhole_5925 := [[447.51, -38.14, 181.08], [0.059327, 0.704614, 0.703506, 0.071266], [0,0,0,0], [9E9, 9E9, 9E9, 9E9, 9E9, 9E9]];
	VAR robtarget Openhole_5926 := [[447.02, -38.07, 181], [0.057416, 0.704772, 0.703365, 0.072646], [0,0,0,0], [9E9, 9E9, 9E9, 9E9, 9E9, 9E9]];
	VAR robtarget Openhole_5927 := [[446.06, -37.84, 180.83], [0.053406, 0.705087, 0.703104, 0.075135], [0,0,0,0], [9E9, 9E9, 9E9, 9E9, 9E9, 9E9]];
	VAR robtarget Openhole_5928 := [[445.11, -37.59, 180.66], [0.049319, 0.705385, 0.702846, 0.077507], [0,0,0,0], [9E9, 9E9, 9E9, 9E9, 9E9, 9E9]];
	VAR robtarget Openhole_5929 := [[444.14, -37.38, 180.5], [0.045342, 0.705652, 0.70256, 0.080059], [0,0,0,0], [9E9, 9E9, 9E9, 9E9, 9E9, 9E9]];
	VAR robtarget Openhole_5930 := [[443.17, -37.22, 180.34], [0.041479, 0.705889, 0.702245, 0.082775], [0,0,0,0], [9E9, 9E9, 9E9, 9E9, 9E9, 9E9]];
	VAR robtarget Openhole_5931 := [[442.19, -37.1, 180.18], [0.037719, 0.7061, 0.701904, 0.085622], [0,0,0,0], [9E9, 9E9, 9E9, 9E9, 9E9, 9E9]];
	VAR robtarget Openhole_5932 := [[438.25, -36.86, 179.52], [0.023449, 0.706718, 0.700309, 0.097812], [0,0,0,0], [9E9, 9E9, 9E9, 9E9, 9E9, 9E9]];
	VAR robtarget Openhole_5933 := [[437.76, -36.86, 179.43], [0.021759, 0.706772, 0.700083, 0.099419], [0,0,0,0], [9E9, 9E9, 9E9, 9E9, 9E9, 9E9]];
	VAR robtarget Openhole_5934 := [[437.27, -36.86, 179.35], [0.020074, 0.706822, 0.699853, 0.101026], [0,0,0,0], [9E9, 9E9, 9E9, 9E9, 9E9, 9E9]];
	VAR robtarget Openhole_5935 := [[429.9, -37.22, 178.02], [-0.003964, 0.707096, 0.69585, 0.125672], [0,0,0,0], [9E9, 9E9, 9E9, 9E9, 9E9, 9E9]];
	VAR robtarget Openhole_5936 := [[424, -37.4, 176.94], [-0.023272, 0.706724, 0.692214, 0.14436], [0,0,0,0], [9E9, 9E9, 9E9, 9E9, 9E9, 9E9]];
	VAR robtarget Openhole_5937 := [[423.51, -37.4, 176.85], [-0.02492, 0.706668, 0.691905, 0.145836], [0,0,0,0], [9E9, 9E9, 9E9, 9E9, 9E9, 9E9]];
	VAR robtarget Openhole_5938 := [[417.59, -37.22, 175.86], [-0.04509, 0.705668, 0.688157, 0.162605], [0,0,0,0], [9E9, 9E9, 9E9, 9E9, 9E9, 9E9]];
	VAR robtarget Openhole_5939 := [[411.68, -36.7, 175.02], [-0.065799, 0.704039, 0.684438, 0.17761], [0,0,0,0], [9E9, 9E9, 9E9, 9E9, 9E9, 9E9]];
	VAR robtarget Openhole_5940 := [[405.77, -35.88, 174.36], [-0.086745, 0.701766, 0.680836, 0.19095], [0,0,0,0], [9E9, 9E9, 9E9, 9E9, 9E9, 9E9]];
	VAR robtarget Openhole_5941 := [[399.88, -34.8, 173.92], [-0.10764, 0.698866, 0.677414, 0.202757], [0,0,0,0], [9E9, 9E9, 9E9, 9E9, 9E9, 9E9]];
	VAR robtarget Openhole_5942 := [[395, -33.77, 173.71], [-0.124731, 0.696019, 0.674682, 0.211669], [0,0,0,0], [9E9, 9E9, 9E9, 9E9, 9E9, 9E9]];
	VAR robtarget Openhole_5943 := [[394.32, -33.65, 173.68], [-0.126951, 0.695617, 0.674278, 0.212953], [0,0,0,0], [9E9, 9E9, 9E9, 9E9, 9E9, 9E9]];
	VAR robtarget Openhole_5944 := [[389.32, -33.65, 172.97], [-0.140659, 0.692975, 0.670532, 0.224471], [0,0,0,0], [9E9, 9E9, 9E9, 9E9, 9E9, 9E9]];
	VAR robtarget Openhole_5945 := [[362.32, -33.65, 173.06], [-0.183051, 0.683002, 0.683002, 0.183051], [0,0,0,0], [9E9, 9E9, 9E9, 9E9, 9E9, 9E9]];
	VAR robtarget Openhole_5946 := [[362.32, -34.53, 172.55], [-0.183051, 0.683002, 0.683002, 0.183051], [0,0,0,0], [9E9, 9E9, 9E9, 9E9, 9E9, 9E9]];
	VAR robtarget Openhole_5947 := [[374.32, -34.53, 172.51], [-0.183051, 0.683002, 0.683002, 0.183051], [0,0,0,0], [9E9, 9E9, 9E9, 9E9, 9E9, 9E9]];
	VAR robtarget Openhole_5948 := [[389.32, -34.53, 172.47], [-0.138176, 0.693475, 0.669724, 0.226869], [0,0,0,0], [9E9, 9E9, 9E9, 9E9, 9E9, 9E9]];
	VAR robtarget Openhole_5949 := [[394.24, -34.53, 173.2], [-0.12465, 0.696033, 0.673434, 0.215609], [0,0,0,0], [9E9, 9E9, 9E9, 9E9, 9E9, 9E9]];
	VAR robtarget Openhole_5950 := [[400.62, -36.11, 173.42], [-0.101564, 0.699775, 0.676832, 0.204692], [0,0,0,0], [9E9, 9E9, 9E9, 9E9, 9E9, 9E9]];
	VAR robtarget Openhole_5951 := [[406, -37.14, 173.87], [-0.08217, 0.702316, 0.679956, 0.194061], [0,0,0,0], [9E9, 9E9, 9E9, 9E9, 9E9, 9E9]];
	VAR robtarget Openhole_5952 := [[412.39, -38.07, 174.65], [-0.05925, 0.70462, 0.683866, 0.179798], [0,0,0,0], [9E9, 9E9, 9E9, 9E9, 9E9, 9E9]];
	VAR robtarget Openhole_5953 := [[418.29, -38.63, 175.57], [-0.038348, 0.706066, 0.687606, 0.164919], [0,0,0,0], [9E9, 9E9, 9E9, 9E9, 9E9, 9E9]];
	VAR robtarget Openhole_5954 := [[418.78, -38.66, 175.65], [-0.036625, 0.706158, 0.68792, 0.163602], [0,0,0,0], [9E9, 9E9, 9E9, 9E9, 9E9, 9E9]];
	VAR robtarget Openhole_5955 := [[419.27, -38.7, 175.73], [-0.034862, 0.706247, 0.688226, 0.162312], [0,0,0,0], [9E9, 9E9, 9E9, 9E9, 9E9, 9E9]];
	VAR robtarget Openhole_5956 := [[408.81, -38.7, 173.75], [-0.068682, 0.703763, 0.68074, 0.191295], [0,0,0,0], [9E9, 9E9, 9E9, 9E9, 9E9, 9E9]];
	VAR robtarget Openhole_5957 := [[408.32, -38.6, 173.7], [-0.070525, 0.703581, 0.680455, 0.192306], [0,0,0,0], [9E9, 9E9, 9E9, 9E9, 9E9, 9E9]];
	VAR robtarget Openhole_5958 := [[402.93, -37.64, 173.11], [-0.090039, 0.701351, 0.677236, 0.203351], [0,0,0,0], [9E9, 9E9, 9E9, 9E9, 9E9, 9E9]];
	VAR robtarget Openhole_5959 := [[398.07, -36.52, 172.8], [-0.107831, 0.698837, 0.674547, 0.212099], [0,0,0,0], [9E9, 9E9, 9E9, 9E9, 9E9, 9E9]];
	VAR robtarget Openhole_5960 := [[395.19, -35.69, 172.74], [-0.118551, 0.697098, 0.673102, 0.216643], [0,0,0,0], [9E9, 9E9, 9E9, 9E9, 9E9, 9E9]];
	VAR robtarget Openhole_5961 := [[394.71, -35.54, 172.74], [-0.120352, 0.696789, 0.672882, 0.217324], [0,0,0,0], [9E9, 9E9, 9E9, 9E9, 9E9, 9E9]];
	VAR robtarget Openhole_5962 := [[394.32, -35.51, 172.7], [-0.121546, 0.696582, 0.672607, 0.218174], [0,0,0,0], [9E9, 9E9, 9E9, 9E9, 9E9, 9E9]];
	VAR robtarget Openhole_5963 := [[389.32, -35.51, 171.9], [-0.135381, 0.694026, 0.668806, 0.229562], [0,0,0,0], [9E9, 9E9, 9E9, 9E9, 9E9, 9E9]];
	VAR robtarget Openhole_5964 := [[360.24, -35.51, 171.99], [-0.183051, 0.683002, 0.683002, 0.183051], [0,0,0,0], [9E9, 9E9, 9E9, 9E9, 9E9, 9E9]];
	VAR robtarget Openhole_5965 := [[360.28, -11.45, 185.89], [-0.183051, 0.683002, 0.683002, 0.183051], [0,0,0,0], [9E9, 9E9, 9E9, 9E9, 9E9, 9E9]];
	VAR robtarget Openhole_5966 := [[389.36, -11.45, 185.8], [-0.203916, 0.677066, 0.688343, 0.161813], [0,0,0,0], [9E9, 9E9, 9E9, 9E9, 9E9, 9E9]];
	VAR robtarget Openhole_5967 := [[394.36, -11.45, 185.43], [-0.1918, 0.680597, 0.691293, 0.148707], [0,0,0,0], [9E9, 9E9, 9E9, 9E9, 9E9, 9E9]];
	VAR robtarget Openhole_5968 := [[406.15, -10.95, 184.78], [-0.162415, 0.688202, 0.697844, 0.114077], [0,0,0,0], [9E9, 9E9, 9E9, 9E9, 9E9, 9E9]];
	VAR robtarget Openhole_5969 := [[427.09, -10.18, 183.32], [-0.102632, 0.699619, 0.705606, 0.046043], [0,0,0,0], [9E9, 9E9, 9E9, 9E9, 9E9, 9E9]];
	VAR robtarget Openhole_5970 := [[441.52, -9.59, 182.13], [-0.057308, 0.704781, 0.707093, -0.004431], [0,0,0,0], [9E9, 9E9, 9E9, 9E9, 9E9, 9E9]];
	VAR robtarget Openhole_5971 := [[443.51, -9.49, 181.96], [-0.050914, 0.705271, 0.707013, -0.011505], [0,0,0,0], [9E9, 9E9, 9E9, 9E9, 9E9, 9E9]];
	VAR robtarget Openhole_5972 := [[445.01, -9.52, 181.82], [-0.045793, 0.705622, 0.706914, -0.016516], [0,0,0,0], [9E9, 9E9, 9E9, 9E9, 9E9, 9E9]];
	VAR robtarget Openhole_5973 := [[447, -9.62, 181.63], [-0.038709, 0.706046, 0.706734, -0.022943], [0,0,0,0], [9E9, 9E9, 9E9, 9E9, 9E9, 9E9]];
	VAR robtarget Openhole_5974 := [[450.48, -9.77, 181.32], [-0.026342, 0.706616, 0.706276, -0.034258], [0,0,0,0], [9E9, 9E9, 9E9, 9E9, 9E9, 9E9]];
	VAR robtarget Openhole_5975 := [[451.47, -9.76, 181.23], [-0.022988, 0.706733, 0.706102, -0.037675], [0,0,0,0], [9E9, 9E9, 9E9, 9E9, 9E9, 9E9]];
	VAR robtarget Openhole_5976 := [[452.97, -9.66, 181.1], [-0.018228, 0.706872, 0.705796, -0.043043], [0,0,0,0], [9E9, 9E9, 9E9, 9E9, 9E9, 9E9]];
	VAR robtarget Openhole_5977 := [[453.46, -9.61, 181.05], [-0.016692, 0.70691, 0.705682, -0.044872], [0,0,0,0], [9E9, 9E9, 9E9, 9E9, 9E9, 9E9]];
	VAR robtarget Openhole_5978 := [[453.96, -9.56, 181], [-0.015199, 0.706943, 0.705561, -0.046734], [0,0,0,0], [9E9, 9E9, 9E9, 9E9, 9E9, 9E9]];
	VAR robtarget Openhole_5979 := [[456.91, -9.15, 180.7], [-0.006464, 0.707077, 0.704722, -0.058026], [0,0,0,0], [9E9, 9E9, 9E9, 9E9, 9E9, 9E9]];
	VAR robtarget Openhole_5980 := [[464.72, -7.68, 179.74], [0.015143, 0.706945, 0.701521, -0.088701], [0,0,0,0], [9E9, 9E9, 9E9, 9E9, 9E9, 9E9]];
	VAR robtarget Openhole_5981 := [[471.06, -6.59, 178.82], [0.032853, 0.706343, 0.698092, -0.112547], [0,0,0,0], [9E9, 9E9, 9E9, 9E9, 9E9, 9E9]];
	VAR robtarget Openhole_5982 := [[475.49, -6.13, 178.18], [0.046018, 0.705608, 0.695469, -0.127761], [0,0,0,0], [9E9, 9E9, 9E9, 9E9, 9E9, 9E9]];
	VAR robtarget Openhole_5983 := [[479.94, -5.98, 177.58], [0.060031, 0.704554, 0.692768, -0.141676], [0,0,0,0], [9E9, 9E9, 9E9, 9E9, 9E9, 9E9]];
	VAR robtarget Openhole_5984 := [[480.44, -5.98, 177.52], [0.061632, 0.704416, 0.692467, -0.143143], [0,0,0,0], [9E9, 9E9, 9E9, 9E9, 9E9, 9E9]];
	VAR robtarget Openhole_5985 := [[485.9, -6.15, 176.89], [0.07951, 0.702622, 0.689132, -0.158419], [0,0,0,0], [9E9, 9E9, 9E9, 9E9, 9E9, 9E9]];
	VAR robtarget Openhole_5986 := [[495.33, -6.89, 176.05], [0.110415, 0.698433, 0.683295, -0.181957], [0,0,0,0], [9E9, 9E9, 9E9, 9E9, 9E9, 9E9]];
	VAR robtarget Openhole_5987 := [[501.3, -7.34, 175.57], [0.128869, 0.695265, 0.679424, -0.195914], [0,0,0,0], [9E9, 9E9, 9E9, 9E9, 9E9, 9E9]];
	VAR robtarget Openhole_5988 := [[504.33, -7.39, 175.26], [0.137427, 0.693624, 0.677281, -0.203201], [0,0,0,0], [9E9, 9E9, 9E9, 9E9, 9E9, 9E9]];
	VAR robtarget Openhole_5989 := [[509.33, -7.39, 174.7], [0.183051, 0.683002, 0.683002, -0.183051], [0,0,0,0], [9E9, 9E9, 9E9, 9E9, 9E9, 9E9]];
	VAR robtarget Openhole_5990 := [[536.33, -7.39, 174.62], [0.183051, 0.683002, 0.683002, -0.183051], [0,0,0,0], [9E9, 9E9, 9E9, 9E9, 9E9, 9E9]];
	VAR robtarget Openhole_5991 := [[536.32, -6.51, 174.11], [0.183051, 0.683002, 0.683002, -0.183051], [0,0,0,0], [9E9, 9E9, 9E9, 9E9, 9E9, 9E9]];
	VAR robtarget Openhole_5992 := [[509.32, -6.51, 174.19], [0.183051, 0.683002, 0.683002, -0.183051], [0,0,0,0], [9E9, 9E9, 9E9, 9E9, 9E9, 9E9]];
	VAR robtarget Openhole_5993 := [[504.33, -6.51, 174.79], [0.134842, 0.694131, 0.676521, -0.205715], [0,0,0,0], [9E9, 9E9, 9E9, 9E9, 9E9, 9E9]];
	VAR robtarget Openhole_5994 := [[504.3, -6.51, 174.8], [0.134756, 0.694148, 0.676542, -0.205647], [0,0,0,0], [9E9, 9E9, 9E9, 9E9, 9E9, 9E9]];
	VAR robtarget Openhole_5995 := [[503.8, -6.51, 174.86], [0.133387, 0.694412, 0.676905, -0.20445], [0,0,0,0], [9E9, 9E9, 9E9, 9E9, 9E9, 9E9]];
	VAR robtarget Openhole_5996 := [[498.83, -6.2, 175.31], [0.118489, 0.697109, 0.680251, -0.193024], [0,0,0,0], [9E9, 9E9, 9E9, 9E9, 9E9, 9E9]];
	VAR robtarget Openhole_5997 := [[488.43, -5.09, 176.18], [0.084048, 0.702094, 0.686676, -0.168748], [0,0,0,0], [9E9, 9E9, 9E9, 9E9, 9E9, 9E9]];
	VAR robtarget Openhole_5998 := [[481.98, -4.67, 176.91], [0.062408, 0.704347, 0.690628, -0.151768], [0,0,0,0], [9E9, 9E9, 9E9, 9E9, 9E9, 9E9]];
	VAR robtarget Openhole_5999 := [[478.51, -4.61, 177.37], [0.051004, 0.705265, 0.692755, -0.141742], [0,0,0,0], [9E9, 9E9, 9E9, 9E9, 9E9, 9E9]];
	VAR robtarget Openhole_6000 := [[478.02, -4.61, 177.44], [0.0494, 0.705379, 0.693058, -0.140251], [0,0,0,0], [9E9, 9E9, 9E9, 9E9, 9E9, 9E9]];
	VAR robtarget Openhole_6001 := [[473.08, -4.83, 178.18], [0.033796, 0.706299, 0.696051, -0.12455], [0,0,0,0], [9E9, 9E9, 9E9, 9E9, 9E9, 9E9]];
	VAR robtarget Openhole_6002 := [[466.7, -5.54, 179.17], [0.014715, 0.706954, 0.699693, -0.102129], [0,0,0,0], [9E9, 9E9, 9E9, 9E9, 9E9, 9E9]];
	VAR robtarget Openhole_6003 := [[463.75, -5.92, 179.6], [0.006006, 0.707081, 0.701179, -0.091365], [0,0,0,0], [9E9, 9E9, 9E9, 9E9, 9E9, 9E9]];
	VAR robtarget Openhole_6004 := [[461.29, -6.17, 179.94], [-0.001532, 0.707105, 0.702282, -0.082465], [0,0,0,0], [9E9, 9E9, 9E9, 9E9, 9E9, 9E9]];
	VAR robtarget Openhole_6005 := [[460.3, -6.24, 180.07], [-0.004676, 0.707091, 0.702682, -0.078979], [0,0,0,0], [9E9, 9E9, 9E9, 9E9, 9E9, 9E9]];
	VAR robtarget Openhole_6006 := [[459.31, -6.28, 180.2], [-0.007918, 0.707062, 0.703058, -0.075562], [0,0,0,0], [9E9, 9E9, 9E9, 9E9, 9E9, 9E9]];
	VAR robtarget Openhole_6007 := [[458.32, -6.3, 180.32], [-0.011254, 0.707017, 0.703409, -0.072218], [0,0,0,0], [9E9, 9E9, 9E9, 9E9, 9E9, 9E9]];
	VAR robtarget Openhole_6008 := [[457.82, -6.3, 180.38], [-0.012956, 0.706988, 0.703576, -0.070572], [0,0,0,0], [9E9, 9E9, 9E9, 9E9, 9E9, 9E9]];
	VAR robtarget Openhole_6009 := [[457.32, -6.28, 180.44], [-0.0147, 0.706954, 0.703735, -0.068968], [0,0,0,0], [9E9, 9E9, 9E9, 9E9, 9E9, 9E9]];
	VAR robtarget Openhole_6010 := [[452.38, -5.84, 181.04], [-0.033088, 0.706332, 0.705052, -0.053863], [0,0,0,0], [9E9, 9E9, 9E9, 9E9, 9E9, 9E9]];
	VAR robtarget Openhole_6011 := [[450.41, -5.64, 181.28], [-0.040506, 0.705946, 0.705485, -0.047871], [0,0,0,0], [9E9, 9E9, 9E9, 9E9, 9E9, 9E9]];
	VAR robtarget Openhole_6012 := [[448.92, -5.55, 181.48], [-0.045856, 0.705618, 0.70579, -0.043128], [0,0,0,0], [9E9, 9E9, 9E9, 9E9, 9E9, 9E9]];
	VAR robtarget Openhole_6013 := [[448.42, -5.54, 181.54], [-0.04757, 0.705505, 0.705889, -0.041474], [0,0,0,0], [9E9, 9E9, 9E9, 9E9, 9E9, 9E9]];
	VAR robtarget Openhole_6014 := [[447.93, -5.54, 181.61], [-0.049243, 0.70539, 0.705987, -0.039778], [0,0,0,0], [9E9, 9E9, 9E9, 9E9, 9E9, 9E9]];
	VAR robtarget Openhole_6015 := [[447.43, -5.56, 181.67], [-0.050851, 0.705276, 0.706084, -0.038021], [0,0,0,0], [9E9, 9E9, 9E9, 9E9, 9E9, 9E9]];
	VAR robtarget Openhole_6016 := [[446.94, -5.6, 181.73], [-0.052404, 0.705162, 0.706179, -0.036215], [0,0,0,0], [9E9, 9E9, 9E9, 9E9, 9E9, 9E9]];
	VAR robtarget Openhole_6017 := [[446.45, -5.65, 181.8], [-0.053913, 0.705048, 0.706271, -0.034373], [0,0,0,0], [9E9, 9E9, 9E9, 9E9, 9E9, 9E9]];
	VAR robtarget Openhole_6018 := [[445.46, -5.78, 181.92], [-0.056821, 0.70482, 0.706444, -0.030599], [0,0,0,0], [9E9, 9E9, 9E9, 9E9, 9E9, 9E9]];
	VAR robtarget Openhole_6019 := [[437.62, -7.11, 182.77], [-0.0786, 0.702725, 0.707107, 0.000554], [0,0,0,0], [9E9, 9E9, 9E9, 9E9, 9E9, 9E9]];
	VAR robtarget Openhole_6020 := [[429.71, -8.01, 183.51], [-0.101411, 0.699797, 0.706462, 0.030194], [0,0,0,0], [9E9, 9E9, 9E9, 9E9, 9E9, 9E9]];
	VAR robtarget Openhole_6021 := [[418.28, -8.88, 184.46], [-0.134019, 0.69429, 0.703597, 0.070367], [0,0,0,0], [9E9, 9E9, 9E9, 9E9, 9E9, 9E9]];
	VAR robtarget Openhole_6022 := [[396.86, -9.88, 186.04], [-0.190106, 0.681072, 0.693651, 0.137289], [0,0,0,0], [9E9, 9E9, 9E9, 9E9, 9E9, 9E9]];
	VAR robtarget Openhole_6023 := [[394.36, -10.02, 186.19], [-0.195915, 0.679424, 0.692179, 0.144528], [0,0,0,0], [9E9, 9E9, 9E9, 9E9, 9E9, 9E9]];
	VAR robtarget Openhole_6024 := [[389.36, -10.02, 186.62], [-0.207927, 0.675845, 0.68929, 0.157733], [0,0,0,0], [9E9, 9E9, 9E9, 9E9, 9E9, 9E9]];
	VAR robtarget Openhole_6025 := [[362.36, -10.02, 186.71], [-0.183051, 0.683002, 0.683002, 0.183051], [0,0,0,0], [9E9, 9E9, 9E9, 9E9, 9E9, 9E9]];
	VAR robtarget Openhole_6026 := [[362.36, -9.02, 187.28], [-0.183051, 0.683002, 0.683002, 0.183051], [0,0,0,0], [9E9, 9E9, 9E9, 9E9, 9E9, 9E9]];
	VAR robtarget Openhole_6027 := [[389.36, -9.02, 187.2], [-0.210728, 0.674977, 0.689937, 0.154878], [0,0,0,0], [9E9, 9E9, 9E9, 9E9, 9E9, 9E9]];
	VAR robtarget Openhole_6028 := [[394.36, -9.02, 186.72], [-0.198789, 0.678589, 0.692783, 0.141603], [0,0,0,0], [9E9, 9E9, 9E9, 9E9, 9E9, 9E9]];
	VAR robtarget Openhole_6029 := [[414.68, -7.96, 185.11], [-0.147525, 0.691546, 0.7027, 0.078816], [0,0,0,0], [9E9, 9E9, 9E9, 9E9, 9E9, 9E9]];
	VAR robtarget Openhole_6030 := [[424.61, -7.15, 184.25], [-0.120261, 0.696805, 0.705719, 0.044277], [0,0,0,0], [9E9, 9E9, 9E9, 9E9, 9E9, 9E9]];
	VAR robtarget Openhole_6031 := [[432.02, -6.25, 183.55], [-0.099742, 0.700037, 0.706911, 0.01663], [0,0,0,0], [9E9, 9E9, 9E9, 9E9, 9E9, 9E9]];
	VAR robtarget Openhole_6032 := [[438.39, -5.14, 182.89], [-0.082592, 0.702267, 0.707054, -0.008621], [0,0,0,0], [9E9, 9E9, 9E9, 9E9, 9E9, 9E9]];
	VAR robtarget Openhole_6033 := [[446.12, -3.31, 181.91], [-0.062839, 0.704309, 0.705915, -0.041044], [0,0,0,0], [9E9, 9E9, 9E9, 9E9, 9E9, 9E9]];
	VAR robtarget Openhole_6034 := [[447.09, -3.15, 181.77], [-0.06006, 0.704552, 0.70568, -0.044891], [0,0,0,0], [9E9, 9E9, 9E9, 9E9, 9E9, 9E9]];
	VAR robtarget Openhole_6035 := [[447.58, -3.09, 181.69], [-0.058614, 0.704673, 0.705558, -0.046773], [0,0,0,0], [9E9, 9E9, 9E9, 9E9, 9E9, 9E9]];
	VAR robtarget Openhole_6036 := [[448.07, -3.04, 181.62], [-0.057103, 0.704797, 0.705435, -0.048602], [0,0,0,0], [9E9, 9E9, 9E9, 9E9, 9E9, 9E9]];
	VAR robtarget Openhole_6037 := [[448.57, -3, 181.54], [-0.055558, 0.704921, 0.705308, -0.050402], [0,0,0,0], [9E9, 9E9, 9E9, 9E9, 9E9, 9E9]];
	VAR robtarget Openhole_6038 := [[449.06, -3, 181.47], [-0.05389, 0.70505, 0.705186, -0.052089], [0,0,0,0], [9E9, 9E9, 9E9, 9E9, 9E9, 9E9]];
	VAR robtarget Openhole_6039 := [[449.56, -3.01, 181.39], [-0.052167, 0.70518, 0.705063, -0.053721], [0,0,0,0], [9E9, 9E9, 9E9, 9E9, 9E9, 9E9]];
	VAR robtarget Openhole_6040 := [[450.54, -3.1, 181.24], [-0.048514, 0.705441, 0.704826, -0.056752], [0,0,0,0], [9E9, 9E9, 9E9, 9E9, 9E9, 9E9]];
	VAR robtarget Openhole_6041 := [[451.03, -3.16, 181.16], [-0.046633, 0.705567, 0.704707, -0.058202], [0,0,0,0], [9E9, 9E9, 9E9, 9E9, 9E9, 9E9]];
	VAR robtarget Openhole_6042 := [[456.9, -4.06, 180.33], [-0.023574, 0.706714, 0.703124, -0.074948], [0,0,0,0], [9E9, 9E9, 9E9, 9E9, 9E9, 9E9]];
	VAR robtarget Openhole_6043 := [[457.4, -4.11, 180.27], [-0.021721, 0.706773, 0.702965, -0.076422], [0,0,0,0], [9E9, 9E9, 9E9, 9E9, 9E9, 9E9]];
	VAR robtarget Openhole_6044 := [[458.38, -4.18, 180.13], [-0.018091, 0.706875, 0.702629, -0.079454], [0,0,0,0], [9E9, 9E9, 9E9, 9E9, 9E9, 9E9]];
	VAR robtarget Openhole_6045 := [[459.37, -4.22, 179.99], [-0.014573, 0.706957, 0.702266, -0.082597], [0,0,0,0], [9E9, 9E9, 9E9, 9E9, 9E9, 9E9]];
	VAR robtarget Openhole_6046 := [[459.87, -4.23, 179.92], [-0.012856, 0.70699, 0.702075, -0.084207], [0,0,0,0], [9E9, 9E9, 9E9, 9E9, 9E9, 9E9]];
	VAR robtarget Openhole_6047 := [[460.36, -4.23, 179.85], [-0.011164, 0.707019, 0.701877, -0.085837], [0,0,0,0], [9E9, 9E9, 9E9, 9E9, 9E9, 9E9]];
	VAR robtarget Openhole_6048 := [[464.81, -4, 179.18], [0.003213, 0.707099, 0.699844, -0.101085], [0,0,0,0], [9E9, 9E9, 9E9, 9E9, 9E9, 9E9]];
	VAR robtarget Openhole_6049 := [[473.16, -3.27, 177.81], [0.029011, 0.706511, 0.695094, -0.129785], [0,0,0,0], [9E9, 9E9, 9E9, 9E9, 9E9, 9E9]];
	VAR robtarget Openhole_6050 := [[477.6, -3.15, 177.1], [0.043323, 0.705778, 0.692364, -0.143637], [0,0,0,0], [9E9, 9E9, 9E9, 9E9, 9E9, 9E9]];
	VAR robtarget Openhole_6051 := [[478.1, -3.15, 177.03], [0.044948, 0.705677, 0.692058, -0.145107], [0,0,0,0], [9E9, 9E9, 9E9, 9E9, 9E9, 9E9]];
	VAR robtarget Openhole_6052 := [[484.03, -3.38, 176.2], [0.064897, 0.704122, 0.68838, -0.161657], [0,0,0,0], [9E9, 9E9, 9E9, 9E9, 9E9, 9E9]];
	VAR robtarget Openhole_6053 := [[490.46, -3.99, 175.47], [0.086924, 0.701744, 0.68443, -0.177641], [0,0,0,0], [9E9, 9E9, 9E9, 9E9, 9E9, 9E9]];
	VAR robtarget Openhole_6054 := [[501.83, -5.45, 174.56], [0.124792, 0.696008, 0.677433, -0.202695], [0,0,0,0], [9E9, 9E9, 9E9, 9E9, 9E9, 9E9]];
	VAR robtarget Openhole_6055 := [[503.82, -5.61, 174.39], [0.130825, 0.694899, 0.676115, -0.207048], [0,0,0,0], [9E9, 9E9, 9E9, 9E9, 9E9, 9E9]];
	VAR robtarget Openhole_6056 := [[504.32, -5.62, 174.33], [0.132234, 0.694632, 0.675759, -0.208205], [0,0,0,0], [9E9, 9E9, 9E9, 9E9, 9E9, 9E9]];
	VAR robtarget Openhole_6057 := [[509.32, -5.62, 173.68], [0.183051, 0.683002, 0.683002, -0.183051], [0,0,0,0], [9E9, 9E9, 9E9, 9E9, 9E9, 9E9]];
	VAR robtarget Openhole_6058 := [[536.32, -5.62, 173.6], [0.183051, 0.683002, 0.683002, -0.183051], [0,0,0,0], [9E9, 9E9, 9E9, 9E9, 9E9, 9E9]];
	VAR robtarget Openhole_6059 := [[536.32, -4.67, 173.05], [0.183051, 0.683002, 0.683002, -0.183051], [0,0,0,0], [9E9, 9E9, 9E9, 9E9, 9E9, 9E9]];
	VAR robtarget Openhole_6060 := [[509.32, -4.67, 173.13], [0.183051, 0.683002, 0.683002, -0.183051], [0,0,0,0], [9E9, 9E9, 9E9, 9E9, 9E9, 9E9]];
	VAR robtarget Openhole_6061 := [[504.32, -4.67, 173.82], [0.12948, 0.695151, 0.674918, -0.210916], [0,0,0,0], [9E9, 9E9, 9E9, 9E9, 9E9, 9E9]];
	VAR robtarget Openhole_6062 := [[503.48, -4.58, 173.89], [0.12687, 0.695632, 0.675467, -0.209152], [0,0,0,0], [9E9, 9E9, 9E9, 9E9, 9E9, 9E9]];
	VAR robtarget Openhole_6063 := [[501.51, -4.28, 174.01], [0.120412, 0.696779, 0.676663, -0.20525], [0,0,0,0], [9E9, 9E9, 9E9, 9E9, 9E9, 9E9]];
	VAR robtarget Openhole_6064 := [[494.13, -3.03, 174.52], [0.095103, 0.700682, 0.681033, -0.190248], [0,0,0,0], [9E9, 9E9, 9E9, 9E9, 9E9, 9E9]];
	VAR robtarget Openhole_6065 := [[487.72, -2.18, 175.2], [0.072799, 0.703349, 0.684948, -0.175629], [0,0,0,0], [9E9, 9E9, 9E9, 9E9, 9E9, 9E9]];
	VAR robtarget Openhole_6066 := [[481.8, -1.7, 176.01], [0.052378, 0.705164, 0.688663, -0.160449], [0,0,0,0], [9E9, 9E9, 9E9, 9E9, 9E9, 9E9]];
	VAR robtarget Openhole_6067 := [[476.86, -1.55, 176.79], [0.035749, 0.706203, 0.691777, -0.14644], [0,0,0,0], [9E9, 9E9, 9E9, 9E9, 9E9, 9E9]];
	VAR robtarget Openhole_6068 := [[476.37, -1.55, 176.87], [0.034118, 0.706283, 0.692088, -0.144965], [0,0,0,0], [9E9, 9E9, 9E9, 9E9, 9E9, 9E9]];
	VAR robtarget Openhole_6069 := [[470.95, -1.73, 177.82], [0.016612, 0.706912, 0.695449, -0.127871], [0,0,0,0], [9E9, 9E9, 9E9, 9E9, 9E9, 9E9]];
	VAR robtarget Openhole_6070 := [[462.6, -2.3, 179.29], [-0.009919, 0.707037, 0.700073, -0.09949], [0,0,0,0], [9E9, 9E9, 9E9, 9E9, 9E9, 9E9]];
	VAR robtarget Openhole_6071 := [[461.12, -2.32, 179.53], [-0.014901, 0.70695, 0.700752, -0.094584], [0,0,0,0], [9E9, 9E9, 9E9, 9E9, 9E9, 9E9]];
	VAR robtarget Openhole_6072 := [[460.13, -2.3, 179.68], [-0.018345, 0.706869, 0.701173, -0.091411], [0,0,0,0], [9E9, 9E9, 9E9, 9E9, 9E9, 9E9]];
	VAR robtarget Openhole_6073 := [[459.64, -2.28, 179.76], [-0.020102, 0.706821, 0.701374, -0.089856], [0,0,0,0], [9E9, 9E9, 9E9, 9E9, 9E9, 9E9]];
	VAR robtarget Openhole_6074 := [[455.71, -1.86, 180.37], [-0.034959, 0.706242, 0.702767, -0.07822], [0,0,0,0], [9E9, 9E9, 9E9, 9E9, 9E9, 9E9]];
	VAR robtarget Openhole_6075 := [[455.22, -1.78, 180.45], [-0.036883, 0.706144, 0.702919, -0.076844], [0,0,0,0], [9E9, 9E9, 9E9, 9E9, 9E9, 9E9]];
	VAR robtarget Openhole_6076 := [[452.8, -1.31, 180.83], [-0.046735, 0.705561, 0.703607, -0.070266], [0,0,0,0], [9E9, 9E9, 9E9, 9E9, 9E9, 9E9]];
	VAR robtarget Openhole_6077 := [[452.32, -1.2, 180.91], [-0.048748, 0.705424, 0.70373, -0.069019], [0,0,0,0], [9E9, 9E9, 9E9, 9E9, 9E9, 9E9]];
	VAR robtarget Openhole_6078 := [[451.35, -1, 181.07], [-0.052708, 0.70514, 0.70398, -0.066426], [0,0,0,0], [9E9, 9E9, 9E9, 9E9, 9E9, 9E9]];
	VAR robtarget Openhole_6079 := [[450.86, -0.92, 181.16], [-0.054633, 0.704993, 0.704108, -0.065049], [0,0,0,0], [9E9, 9E9, 9E9, 9E9, 9E9, 9E9]];
	VAR robtarget Openhole_6080 := [[450.38, -0.87, 181.24], [-0.056477, 0.704848, 0.704243, -0.06357], [0,0,0,0], [9E9, 9E9, 9E9, 9E9, 9E9, 9E9]];
	VAR robtarget Openhole_6081 := [[449.88, -0.83, 181.33], [-0.058275, 0.704701, 0.70438, -0.062033], [0,0,0,0], [9E9, 9E9, 9E9, 9E9, 9E9, 9E9]];
	VAR robtarget Openhole_6082 := [[449.39, -0.83, 181.41], [-0.059933, 0.704562, 0.704527, -0.060348], [0,0,0,0], [9E9, 9E9, 9E9, 9E9, 9E9, 9E9]];
	VAR robtarget Openhole_6083 := [[448.9, -0.86, 181.5], [-0.061528, 0.704425, 0.704674, -0.058607], [0,0,0,0], [9E9, 9E9, 9E9, 9E9, 9E9, 9E9]];
	VAR robtarget Openhole_6084 := [[448.41, -0.92, 181.58], [-0.062969, 0.704297, 0.704827, -0.056734], [0,0,0,0], [9E9, 9E9, 9E9, 9E9, 9E9, 9E9]];
	VAR robtarget Openhole_6085 := [[447.93, -1.01, 181.67], [-0.064321, 0.704175, 0.70498, -0.054798], [0,0,0,0], [9E9, 9E9, 9E9, 9E9, 9E9, 9E9]];
	VAR robtarget Openhole_6086 := [[447.44, -1.11, 181.75], [-0.065614, 0.704056, 0.705131, -0.052819], [0,0,0,0], [9E9, 9E9, 9E9, 9E9, 9E9, 9E9]];
	VAR robtarget Openhole_6087 := [[446.48, -1.34, 181.91], [-0.068114, 0.703818, 0.70542, -0.048805], [0,0,0,0], [9E9, 9E9, 9E9, 9E9, 9E9, 9E9]];
	VAR robtarget Openhole_6088 := [[438.37, -3.6, 183.05], [-0.087736, 0.701643, 0.706975, -0.013653], [0,0,0,0], [9E9, 9E9, 9E9, 9E9, 9E9, 9E9]];
	VAR robtarget Openhole_6089 := [[433.03, -4.74, 183.67], [-0.101442, 0.699793, 0.707058, 0.008264], [0,0,0,0], [9E9, 9E9, 9E9, 9E9, 9E9, 9E9]];
	VAR robtarget Openhole_6090 := [[426.64, -5.75, 184.32], [-0.118471, 0.697112, 0.706337, 0.03299], [0,0,0,0], [9E9, 9E9, 9E9, 9E9, 9E9, 9E9]];
	VAR robtarget Openhole_6091 := [[418.23, -6.67, 185.12], [-0.141164, 0.692873, 0.704254, 0.063458], [0,0,0,0], [9E9, 9E9, 9E9, 9E9, 9E9, 9E9]];
	VAR robtarget Openhole_6092 := [[406.31, -7.48, 186.21], [-0.172555, 0.685729, 0.699576, 0.102927], [0,0,0,0], [9E9, 9E9, 9E9, 9E9, 9E9, 9E9]];
	VAR robtarget Openhole_6093 := [[394.35, -8.14, 187.19], [-0.201353, 0.677833, 0.693299, 0.139058], [0,0,0,0], [9E9, 9E9, 9E9, 9E9, 9E9, 9E9]];
	VAR robtarget Openhole_6094 := [[389.37, -8.14, 187.71], [-0.213196, 0.674202, 0.690498, 0.152357], [0,0,0,0], [9E9, 9E9, 9E9, 9E9, 9E9, 9E9]];
	VAR robtarget Openhole_6095 := [[362.37, -8.14, 187.79], [-0.183051, 0.683002, 0.683002, 0.183051], [0,0,0,0], [9E9, 9E9, 9E9, 9E9, 9E9, 9E9]];
	VAR robtarget Openhole_6096 := [[362.37, -7.26, 188.3], [-0.183051, 0.683002, 0.683002, 0.183051], [0,0,0,0], [9E9, 9E9, 9E9, 9E9, 9E9, 9E9]];
	VAR robtarget Openhole_6097 := [[374.37, -7.26, 188.27], [-0.183051, 0.683002, 0.683002, 0.183051], [0,0,0,0], [9E9, 9E9, 9E9, 9E9, 9E9, 9E9]];
	VAR robtarget Openhole_6098 := [[389.37, -7.26, 188.22], [-0.215657, 0.673418, 0.691049, 0.149837], [0,0,0,0], [9E9, 9E9, 9E9, 9E9, 9E9, 9E9]];
	VAR robtarget Openhole_6099 := [[394.35, -7.26, 187.65], [-0.203888, 0.677074, 0.693809, 0.136489], [0,0,0,0], [9E9, 9E9, 9E9, 9E9, 9E9, 9E9]];
	VAR robtarget Openhole_6100 := [[412.75, -6.11, 185.97], [-0.158828, 0.689038, 0.702679, 0.079006], [0,0,0,0], [9E9, 9E9, 9E9, 9E9, 9E9, 9E9]];
	VAR robtarget Openhole_6101 := [[421.67, -5.25, 185.09], [-0.135383, 0.694026, 0.705493, 0.047751], [0,0,0,0], [9E9, 9E9, 9E9, 9E9, 9E9, 9E9]];
	VAR robtarget Openhole_6102 := [[429.05, -4.16, 184.33], [-0.116055, 0.697518, 0.706831, 0.019755], [0,0,0,0], [9E9, 9E9, 9E9, 9E9, 9E9, 9E9]];
	VAR robtarget Openhole_6103 := [[435.37, -2.86, 183.6], [-0.100018, 0.699997, 0.707082, -0.00591], [0,0,0,0], [9E9, 9E9, 9E9, 9E9, 9E9, 9E9]];
	VAR robtarget Openhole_6104 := [[442.06, -1.02, 182.68], [-0.083997, 0.7021, 0.70625, -0.034792], [0,0,0,0], [9E9, 9E9, 9E9, 9E9, 9E9, 9E9]];
	VAR robtarget Openhole_6105 := [[446.81, 0.36, 181.9], [-0.072617, 0.703368, 0.704926, -0.055486], [0,0,0,0], [9E9, 9E9, 9E9, 9E9, 9E9, 9E9]];
	VAR robtarget Openhole_6106 := [[447.76, 0.61, 181.72], [-0.070216, 0.703612, 0.704596, -0.059541], [0,0,0,0], [9E9, 9E9, 9E9, 9E9, 9E9, 9E9]];
	VAR robtarget Openhole_6107 := [[448.72, 0.81, 181.54], [-0.067626, 0.703866, 0.704252, -0.063471], [0,0,0,0], [9E9, 9E9, 9E9, 9E9, 9E9, 9E9]];
	VAR robtarget Openhole_6108 := [[449.21, 0.87, 181.45], [-0.06615, 0.704006, 0.704085, -0.065304], [0,0,0,0], [9E9, 9E9, 9E9, 9E9, 9E9, 9E9]];
	VAR robtarget Openhole_6109 := [[449.7, 0.9, 181.35], [-0.064595, 0.70415, 0.703919, -0.067071], [0,0,0,0], [9E9, 9E9, 9E9, 9E9, 9E9, 9E9]];
	VAR robtarget Openhole_6110 := [[450.19, 0.88, 181.26], [-0.062848, 0.704308, 0.703766, -0.068652], [0,0,0,0], [9E9, 9E9, 9E9, 9E9, 9E9, 9E9]];
	VAR robtarget Openhole_6111 := [[450.68, 0.85, 181.17], [-0.061074, 0.704464, 0.703613, -0.0702], [0,0,0,0], [9E9, 9E9, 9E9, 9E9, 9E9, 9E9]];
	VAR robtarget Openhole_6112 := [[451.17, 0.77, 181.07], [-0.059183, 0.704626, 0.703472, -0.071607], [0,0,0,0], [9E9, 9E9, 9E9, 9E9, 9E9, 9E9]];
	VAR robtarget Openhole_6113 := [[451.65, 0.69, 180.98], [-0.057244, 0.704786, 0.703334, -0.072949], [0,0,0,0], [9E9, 9E9, 9E9, 9E9, 9E9, 9E9]];
	VAR robtarget Openhole_6114 := [[453.08, 0.32, 180.73], [-0.051162, 0.705253, 0.702948, -0.076577], [0,0,0,0], [9E9, 9E9, 9E9, 9E9, 9E9, 9E9]];
	VAR robtarget Openhole_6115 := [[453.56, 0.19, 180.64], [-0.049098, 0.7054, 0.702822, -0.077726], [0,0,0,0], [9E9, 9E9, 9E9, 9E9, 9E9, 9E9]];
	VAR robtarget Openhole_6116 := [[454.52, -0.01, 180.47], [-0.045136, 0.705665, 0.702532, -0.080301], [0,0,0,0], [9E9, 9E9, 9E9, 9E9, 9E9, 9E9]];
	VAR robtarget Openhole_6117 := [[455.49, -0.16, 180.3], [-0.041297, 0.7059, 0.702213, -0.083048], [0,0,0,0], [9E9, 9E9, 9E9, 9E9, 9E9, 9E9]];
	VAR robtarget Openhole_6118 := [[456.96, -0.33, 180.05], [-0.035715, 0.706204, 0.701686, -0.087385], [0,0,0,0], [9E9, 9E9, 9E9, 9E9, 9E9, 9E9]];
	VAR robtarget Openhole_6119 := [[457.94, -0.41, 179.88], [-0.032089, 0.706378, 0.701307, -0.09038], [0,0,0,0], [9E9, 9E9, 9E9, 9E9, 9E9, 9E9]];
	VAR robtarget Openhole_6120 := [[459.91, -0.49, 179.54], [-0.025059, 0.706663, 0.70048, -0.096579], [0,0,0,0], [9E9, 9E9, 9E9, 9E9, 9E9, 9E9]];
	VAR robtarget Openhole_6121 := [[460.9, -0.5, 179.36], [-0.021661, 0.706775, 0.700032, -0.099777], [0,0,0,0], [9E9, 9E9, 9E9, 9E9, 9E9, 9E9]];
	VAR robtarget Openhole_6122 := [[467.28, -0.21, 178.17], [-0.00078, 0.707106, 0.696639, -0.121218], [0,0,0,0], [9E9, 9E9, 9E9, 9E9, 9E9, 9E9]];
	VAR robtarget Openhole_6123 := [[474.15, 0.08, 176.86], [0.021502, 0.70678, 0.692416, -0.14339], [0,0,0,0], [9E9, 9E9, 9E9, 9E9, 9E9, 9E9]];
	VAR robtarget Openhole_6124 := [[475.62, 0.08, 176.59], [0.026406, 0.706614, 0.691476, -0.147857], [0,0,0,0], [9E9, 9E9, 9E9, 9E9, 9E9, 9E9]];
	VAR robtarget Openhole_6125 := [[476.12, 0.08, 176.5], [0.028056, 0.70655, 0.691162, -0.149315], [0,0,0,0], [9E9, 9E9, 9E9, 9E9, 9E9, 9E9]];
	VAR robtarget Openhole_6126 := [[482.02, -0.15, 175.48], [0.048239, 0.705459, 0.687381, -0.165853], [0,0,0,0], [9E9, 9E9, 9E9, 9E9, 9E9, 9E9]];
	VAR robtarget Openhole_6127 := [[487.93, -0.71, 174.61], [0.068896, 0.703742, 0.68364, -0.180656], [0,0,0,0], [9E9, 9E9, 9E9, 9E9, 9E9, 9E9]];
	VAR robtarget Openhole_6128 := [[493.83, -1.55, 173.94], [0.089733, 0.70139, 0.680023, -0.193827], [0,0,0,0], [9E9, 9E9, 9E9, 9E9, 9E9, 9E9]];
	VAR robtarget Openhole_6129 := [[499.22, -2.58, 173.52], [0.108824, 0.698683, 0.676893, -0.20449], [0,0,0,0], [9E9, 9E9, 9E9, 9E9, 9E9, 9E9]];
	VAR robtarget Openhole_6130 := [[503.61, -3.55, 173.33], [0.12421, 0.696112, 0.67445, -0.212408], [0,0,0,0], [9E9, 9E9, 9E9, 9E9, 9E9, 9E9]];
	VAR robtarget Openhole_6131 := [[504.32, -3.66, 173.29], [0.126534, 0.695693, 0.674021, -0.213765], [0,0,0,0], [9E9, 9E9, 9E9, 9E9, 9E9, 9E9]];
	VAR robtarget Openhole_6132 := [[509.32, -3.66, 172.55], [0.183051, 0.683002, 0.683002, -0.183051], [0,0,0,0], [9E9, 9E9, 9E9, 9E9, 9E9, 9E9]];
	VAR robtarget Openhole_6133 := [[536.32, -3.66, 172.46], [0.183051, 0.683002, 0.683002, -0.183051], [0,0,0,0], [9E9, 9E9, 9E9, 9E9, 9E9, 9E9]];
	VAR robtarget Openhole_6134 := [[536.32, -2.79, 171.96], [0.183051, 0.683002, 0.683002, -0.183051], [0,0,0,0], [9E9, 9E9, 9E9, 9E9, 9E9, 9E9]];
	VAR robtarget Openhole_6135 := [[524.32, -2.79, 172], [0.183051, 0.683002, 0.683002, -0.183051], [0,0,0,0], [9E9, 9E9, 9E9, 9E9, 9E9, 9E9]];
	VAR robtarget Openhole_6136 := [[509.32, -2.79, 172.05], [0.183051, 0.683002, 0.683002, -0.183051], [0,0,0,0], [9E9, 9E9, 9E9, 9E9, 9E9, 9E9]];
	VAR robtarget Openhole_6137 := [[504.4, -2.79, 172.81], [0.12423, 0.696108, 0.673175, -0.216414], [0,0,0,0], [9E9, 9E9, 9E9, 9E9, 9E9, 9E9]];
	VAR robtarget Openhole_6138 := [[503.83, -2.67, 172.84], [0.12228, 0.696454, 0.673499, -0.215406], [0,0,0,0], [9E9, 9E9, 9E9, 9E9, 9E9, 9E9]];
	VAR robtarget Openhole_6139 := [[498.02, -1.2, 173.07], [0.101197, 0.699828, 0.676588, -0.205497], [0,0,0,0], [9E9, 9E9, 9E9, 9E9, 9E9, 9E9]];
	VAR robtarget Openhole_6140 := [[492.65, -0.16, 173.55], [0.081862, 0.702352, 0.679732, -0.194845], [0,0,0,0], [9E9, 9E9, 9E9, 9E9, 9E9, 9E9]];
	VAR robtarget Openhole_6141 := [[486.76, 0.7, 174.32], [0.060823, 0.704486, 0.683375, -0.181654], [0,0,0,0], [9E9, 9E9, 9E9, 9E9, 9E9, 9E9]];
	VAR robtarget Openhole_6142 := [[480.86, 1.26, 175.26], [0.03999, 0.705975, 0.68714, -0.166849], [0,0,0,0], [9E9, 9E9, 9E9, 9E9, 9E9, 9E9]];
	VAR robtarget Openhole_6143 := [[480.37, 1.3, 175.35], [0.038253, 0.706071, 0.687453, -0.165556], [0,0,0,0], [9E9, 9E9, 9E9, 9E9, 9E9, 9E9]];
	VAR robtarget Openhole_6144 := [[490.33, 1.3, 173.4], [0.070258, 0.703608, 0.680237, -0.193073], [0,0,0,0], [9E9, 9E9, 9E9, 9E9, 9E9, 9E9]];
	VAR robtarget Openhole_6145 := [[490.83, 1.18, 173.35], [0.072176, 0.703414, 0.679971, -0.19401], [0,0,0,0], [9E9, 9E9, 9E9, 9E9, 9E9, 9E9]];
	VAR robtarget Openhole_6146 := [[496.2, 0.2, 172.74], [0.091597, 0.701149, 0.67674, -0.204996], [0,0,0,0], [9E9, 9E9, 9E9, 9E9, 9E9, 9E9]];
	VAR robtarget Openhole_6147 := [[501.06, -0.96, 172.42], [0.109345, 0.698601, 0.674067, -0.213622], [0,0,0,0], [9E9, 9E9, 9E9, 9E9, 9E9, 9E9]];
	VAR robtarget Openhole_6148 := [[502.98, -1.51, 172.38], [0.116483, 0.697447, 0.673103, -0.216639], [0,0,0,0], [9E9, 9E9, 9E9, 9E9, 9E9, 9E9]];
	VAR robtarget Openhole_6149 := [[503.45, -1.68, 172.38], [0.118298, 0.697141, 0.672889, -0.217301], [0,0,0,0], [9E9, 9E9, 9E9, 9E9, 9E9, 9E9]];
	VAR robtarget Openhole_6150 := [[504.32, -1.86, 172.34], [0.121295, 0.696626, 0.672398, -0.218816], [0,0,0,0], [9E9, 9E9, 9E9, 9E9, 9E9, 9E9]];
	VAR robtarget Openhole_6151 := [[509.32, -1.86, 171.51], [0.183051, 0.683002, 0.683002, -0.183051], [0,0,0,0], [9E9, 9E9, 9E9, 9E9, 9E9, 9E9]];
	VAR robtarget Openhole_6152 := [[536.32, -1.86, 171.43], [0.183051, 0.683002, 0.683002, -0.183051], [0,0,0,0], [9E9, 9E9, 9E9, 9E9, 9E9, 9E9]];
	VAR robtarget Openhole_6153 := [[536.31, -1.34, 171.12], [0.183051, 0.683002, 0.683002, -0.183051], [0,0,0,0], [9E9, 9E9, 9E9, 9E9, 9E9, 9E9]];
	VAR robtarget Openhole_6154 := [[509.31, -1.34, 171.21], [0.183051, 0.683002, 0.683002, -0.183051], [0,0,0,0], [9E9, 9E9, 9E9, 9E9, 9E9, 9E9]];
	VAR robtarget Openhole_6155 := [[504.32, -1.34, 172.06], [0.119767, 0.69689, 0.671918, -0.220286], [0,0,0,0], [9E9, 9E9, 9E9, 9E9, 9E9, 9E9]];
	VAR robtarget Openhole_6156 := [[503.61, -1.18, 172.09], [0.117291, 0.697311, 0.672314, -0.219074], [0,0,0,0], [9E9, 9E9, 9E9, 9E9, 9E9, 9E9]];
	VAR robtarget Openhole_6157 := [[499.76, -0.1, 172.23], [0.103043, 0.699558, 0.674291, -0.212912], [0,0,0,0], [9E9, 9E9, 9E9, 9E9, 9E9, 9E9]];
	VAR robtarget Openhole_6158 := [[494.89, 0.95, 172.66], [0.085371, 0.701934, 0.677085, -0.203852], [0,0,0,0], [9E9, 9E9, 9E9, 9E9, 9E9, 9E9]];
	VAR robtarget Openhole_6159 := [[492.93, 1.3, 172.89], [0.078335, 0.702754, 0.678274, -0.199862], [0,0,0,0], [9E9, 9E9, 9E9, 9E9, 9E9, 9E9]];
	VAR robtarget Openhole_6160 := [[445.28, 1.3, 182.22], [-0.080802, 0.702475, 0.705092, -0.053344], [0,0,0,0], [9E9, 9E9, 9E9, 9E9, 9E9, 9E9]];
	VAR robtarget Openhole_6161 := [[444.81, 1.13, 182.3], [-0.081872, 0.702351, 0.70525, -0.051214], [0,0,0,0], [9E9, 9E9, 9E9, 9E9, 9E9, 9E9]];
	VAR robtarget Openhole_6162 := [[436.71, -1.11, 183.6], [-0.10136, 0.699804, 0.706921, -0.01622], [0,0,0,0], [9E9, 9E9, 9E9, 9E9, 9E9, 9E9]];
	VAR robtarget Openhole_6163 := [[429.96, -2.73, 184.46], [-0.117791, 0.697227, 0.707005, 0.012025], [0,0,0,0], [9E9, 9E9, 9E9, 9E9, 9E9, 9E9]];
	VAR robtarget Openhole_6164 := [[423.11, -3.95, 185.23], [-0.135135, 0.694074, 0.70604, 0.038834], [0,0,0,0], [9E9, 9E9, 9E9, 9E9, 9E9, 9E9]];
	VAR robtarget Openhole_6165 := [[415.71, -4.87, 186.01], [-0.154221, 0.690084, 0.704042, 0.065763], [0,0,0,0], [9E9, 9E9, 9E9, 9E9, 9E9, 9E9]];
	VAR robtarget Openhole_6166 := [[405.3, -5.7, 187.08], [-0.180626, 0.683648, 0.69993, 0.100488], [0,0,0,0], [9E9, 9E9, 9E9, 9E9, 9E9, 9E9]];
	VAR robtarget Openhole_6167 := [[394.35, -6.37, 188.12], [-0.206401, 0.676313, 0.694313, 0.133901], [0,0,0,0], [9E9, 9E9, 9E9, 9E9, 9E9, 9E9]];
	VAR robtarget Openhole_6168 := [[389.37, -6.37, 188.73], [-0.218114, 0.672627, 0.691591, 0.147317], [0,0,0,0], [9E9, 9E9, 9E9, 9E9, 9E9, 9E9]];
	VAR robtarget Openhole_6169 := [[362.37, -6.37, 188.81], [-0.183051, 0.683002, 0.683002, 0.183051], [0,0,0,0], [9E9, 9E9, 9E9, 9E9, 9E9, 9E9]];
	VAR robtarget Openhole_6170 := [[362.37, -5.47, 189.34], [-0.183051, 0.683002, 0.683002, 0.183051], [0,0,0,0], [9E9, 9E9, 9E9, 9E9, 9E9, 9E9]];
	VAR robtarget Openhole_6171 := [[389.37, -5.47, 189.25], [-0.220622, 0.671808, 0.692135, 0.144739], [0,0,0,0], [9E9, 9E9, 9E9, 9E9, 9E9, 9E9]];
	VAR robtarget Openhole_6172 := [[394.37, -5.47, 188.6], [-0.208939, 0.675533, 0.694825, 0.131219], [0,0,0,0], [9E9, 9E9, 9E9, 9E9, 9E9, 9E9]];
	VAR robtarget Openhole_6173 := [[410.22, -4.4, 186.93], [-0.171212, 0.686066, 0.702392, 0.081519], [0,0,0,0], [9E9, 9E9, 9E9, 9E9, 9E9, 9E9]];
	VAR robtarget Openhole_6174 := [[418.62, -3.5, 186.02], [-0.150001, 0.691014, 0.705187, 0.052073], [0,0,0,0], [9E9, 9E9, 9E9, 9E9, 9E9, 9E9]];
	VAR robtarget Openhole_6175 := [[425, -2.5, 185.3], [-0.133982, 0.694297, 0.706556, 0.027897], [0,0,0,0], [9E9, 9E9, 9E9, 9E9, 9E9, 9E9]];
	VAR robtarget Openhole_6176 := [[431.79, -1.04, 184.46], [-0.117445, 0.697285, 0.707107, 0.000297], [0,0,0,0], [9E9, 9E9, 9E9, 9E9, 9E9, 9E9]];
	VAR robtarget Openhole_6177 := [[440.43, 1.14, 183.15], [-0.09649, 0.700492, 0.706176, -0.036272], [0,0,0,0], [9E9, 9E9, 9E9, 9E9, 9E9, 9E9]];
	VAR robtarget Openhole_6178 := [[440.9, 1.3, 183.07], [-0.095371, 0.700646, 0.706065, -0.038361], [0,0,0,0], [9E9, 9E9, 9E9, 9E9, 9E9, 9E9]];
	VAR robtarget Openhole_6179 := [[436.08, 1.3, 184.02], [-0.111136, 0.698319, 0.70677, -0.021814], [0,0,0,0], [9E9, 9E9, 9E9, 9E9, 9E9, 9E9]];
	VAR robtarget Openhole_6180 := [[435.6, 1.08, 184.08], [-0.112081, 0.698168, 0.706836, -0.01955], [0,0,0,0], [9E9, 9E9, 9E9, 9E9, 9E9, 9E9]];
	VAR robtarget Openhole_6181 := [[427.41, -0.87, 185.26], [-0.131755, 0.694723, 0.706957, 0.014576], [0,0,0,0], [9E9, 9E9, 9E9, 9E9, 9E9, 9E9]];
	VAR robtarget Openhole_6182 := [[420.58, -2.17, 186.09], [-0.148386, 0.691362, 0.705892, 0.041425], [0,0,0,0], [9E9, 9E9, 9E9, 9E9, 9E9, 9E9]];
	VAR robtarget Openhole_6183 := [[413.2, -3.14, 186.95], [-0.166738, 0.687167, 0.703801, 0.068299], [0,0,0,0], [9E9, 9E9, 9E9, 9E9, 9E9, 9E9]];
	VAR robtarget Openhole_6184 := [[403.3, -3.99, 188.09], [-0.190959, 0.680834, 0.69982, 0.101252], [0,0,0,0], [9E9, 9E9, 9E9, 9E9, 9E9, 9E9]];
	VAR robtarget Openhole_6185 := [[394.36, -4.59, 189.07], [-0.21147, 0.674745, 0.6953, 0.128677], [0,0,0,0], [9E9, 9E9, 9E9, 9E9, 9E9, 9E9]];
	VAR robtarget Openhole_6186 := [[389.37, -4.59, 189.76], [-0.223064, 0.671001, 0.692656, 0.142225], [0,0,0,0], [9E9, 9E9, 9E9, 9E9, 9E9, 9E9]];
	VAR robtarget Openhole_6187 := [[362.37, -4.58, 189.85], [-0.183051, 0.683002, 0.683002, 0.183051], [0,0,0,0], [9E9, 9E9, 9E9, 9E9, 9E9, 9E9]];
	VAR robtarget Openhole_6188 := [[362.37, -3.7, 190.36], [-0.183051, 0.683002, 0.683002, 0.183051], [0,0,0,0], [9E9, 9E9, 9E9, 9E9, 9E9, 9E9]];
	VAR robtarget Openhole_6189 := [[374.37, -3.7, 190.32], [-0.183051, 0.683002, 0.683002, 0.183051], [0,0,0,0], [9E9, 9E9, 9E9, 9E9, 9E9, 9E9]];
	VAR robtarget Openhole_6190 := [[389.37, -3.7, 190.27], [-0.2255, 0.670186, 0.693167, 0.139712], [0,0,0,0], [9E9, 9E9, 9E9, 9E9, 9E9, 9E9]];
	VAR robtarget Openhole_6191 := [[394.37, -3.7, 189.53], [-0.213956, 0.673961, 0.695774, 0.126089], [0,0,0,0], [9E9, 9E9, 9E9, 9E9, 9E9, 9E9]];
	VAR robtarget Openhole_6192 := [[408.73, -2.65, 187.83], [-0.18057, 0.683663, 0.702486, 0.080703], [0,0,0,0], [9E9, 9E9, 9E9, 9E9, 9E9, 9E9]];
	VAR robtarget Openhole_6193 := [[416.62, -1.76, 186.86], [-0.161246, 0.688476, 0.705118, 0.053001], [0,0,0,0], [9E9, 9E9, 9E9, 9E9, 9E9, 9E9]];
	VAR robtarget Openhole_6194 := [[423.48, -0.63, 186], [-0.144526, 0.692179, 0.706592, 0.026964], [0,0,0,0], [9E9, 9E9, 9E9, 9E9, 9E9, 9E9]];
	VAR robtarget Openhole_6195 := [[430.74, 0.96, 185], [-0.127188, 0.695574, 0.707102, -0.002584], [0,0,0,0], [9E9, 9E9, 9E9, 9E9, 9E9, 9E9]];
	VAR robtarget Openhole_6196 := [[431.22, 1.07, 184.93], [-0.126041, 0.695783, 0.707092, -0.004593], [0,0,0,0], [9E9, 9E9, 9E9, 9E9, 9E9, 9E9]];
	VAR robtarget Openhole_6197 := [[431.7, 1.3, 184.88], [-0.125115, 0.69595, 0.707074, -0.006843], [0,0,0,0], [9E9, 9E9, 9E9, 9E9, 9E9, 9E9]];
	VAR robtarget Openhole_6198 := [[427.8, 1.3, 185.64], [-0.137278, 0.693653, 0.707078, 0.006418], [0,0,0,0], [9E9, 9E9, 9E9, 9E9, 9E9, 9E9]];
	VAR robtarget Openhole_6199 := [[427.32, 1.15, 185.7], [-0.138449, 0.69342, 0.707057, 0.008373], [0,0,0,0], [9E9, 9E9, 9E9, 9E9, 9E9, 9E9]];
	VAR robtarget Openhole_6200 := [[420.52, -0.2, 186.65], [-0.154723, 0.689972, 0.706221, 0.035383], [0,0,0,0], [9E9, 9E9, 9E9, 9E9, 9E9, 9E9]];
	VAR robtarget Openhole_6201 := [[413.16, -1.26, 187.61], [-0.172597, 0.685719, 0.704334, 0.062558], [0,0,0,0], [9E9, 9E9, 9E9, 9E9, 9E9, 9E9]];
	VAR robtarget Openhole_6202 := [[404.27, -2.12, 188.76], [-0.19394, 0.679991, 0.701004, 0.092703], [0,0,0,0], [9E9, 9E9, 9E9, 9E9, 9E9, 9E9]];
	VAR robtarget Openhole_6203 := [[394.37, -2.82, 190], [-0.21644, 0.673167, 0.696236, 0.123511], [0,0,0,0], [9E9, 9E9, 9E9, 9E9, 9E9, 9E9]];
	VAR robtarget Openhole_6204 := [[389.38, -2.82, 190.78], [-0.227928, 0.669364, 0.693668, 0.137201], [0,0,0,0], [9E9, 9E9, 9E9, 9E9, 9E9, 9E9]];
	VAR robtarget Openhole_6205 := [[362.38, -2.82, 190.87], [-0.183051, 0.683002, 0.683002, 0.183051], [0,0,0,0], [9E9, 9E9, 9E9, 9E9, 9E9, 9E9]];
	VAR robtarget Openhole_6206 := [[362.38, -1.93, 191.38], [-0.183051, 0.683002, 0.683002, 0.183051], [0,0,0,0], [9E9, 9E9, 9E9, 9E9, 9E9, 9E9]];
	VAR robtarget Openhole_6207 := [[389.38, -1.93, 191.29], [-0.230349, 0.668535, 0.69416, 0.134694], [0,0,0,0], [9E9, 9E9, 9E9, 9E9, 9E9, 9E9]];
	VAR robtarget Openhole_6208 := [[394.37, -1.93, 190.47], [-0.218917, 0.672366, 0.696688, 0.120937], [0,0,0,0], [9E9, 9E9, 9E9, 9E9, 9E9, 9E9]];
	VAR robtarget Openhole_6209 := [[406.73, -1.02, 188.81], [-0.190765, 0.680888, 0.702348, 0.081896], [0,0,0,0], [9E9, 9E9, 9E9, 9E9, 9E9, 9E9]];
	VAR robtarget Openhole_6210 := [[415.1, -0.08, 187.67], [-0.170727, 0.686187, 0.705143, 0.052666], [0,0,0,0], [9E9, 9E9, 9E9, 9E9, 9E9, 9E9]];
	VAR robtarget Openhole_6211 := [[422.43, 1.1, 186.64], [-0.153078, 0.690338, 0.706667, 0.024924], [0,0,0,0], [9E9, 9E9, 9E9, 9E9, 9E9, 9E9]];
